// SIMATIC STEP 7 (V5.x) project MK2105
// CPU: CPU 317F-3 PN/DP
// station: 硬件
// station: SINUMERIK
// station: P_ADR_BUS
// program: S7 程序
// program: SINAMICS_In_NCU_710

SYMBOL_TABLE
"ALMSG_DB"	DB 2	UDT 2	// Interface for Alarms & Messages
"gp_par"	DB 7	FB 1	// Parameters for Baseprogram
"NC"	DB 10	UDT 10	// Interface NC
"BAG"	DB 11	UDT 11	// Interface for BAG
"PI"	DB 16	DB 16	// Datainterface PI-Services
"SPL"	DB 18	DB 18	// SPL dataarea
"MMC"	DB 19	UDT 19	// Interface MMC-Signals
"Chan1"	DB 21	UDT 21	// Interface for Channel 1
"X"	DB 31	UDT 31	// Interface Axis 1
"Z"	DB 32	UDT 31	// Interface Axis 2
"C"	DB 33	UDT 31	// Interface Axis 3
"A"	DB 34	UDT 31	// Interface Axis 4
"V"	DB 35	UDT 31	// Interface Axis 5
"W"	DB 36	UDT 31	// Interface Axis 6
"TMLoadIF"	DB 71	UDT 71	// Interface for Loading Station (Toolmanag.)
"TMSpindleIF"	DB 72	UDT 72	// Interface Spindle for Toolmanagment
"TMRevIF"	DB 73	UDT 73	// Interface Revolver (Toolmanagment)
"READ_DB0"	DB 100	DB 100	// Read nc data block0
"READ_DB2"	DB 102	DB 102	// Read nc data R296----R299
"Program_Select"	DB 103	DB 103	// Save PLC Select SUB Programe name
"READ_DB3"	DB 104	DB 104	// Read nc data block3
"X_BACK"	DB 106	DB 106	// X_BACK
"SYSTEM_DB"	DB 110	DB 110	// Read system date and time
"USER_DB0"	DB 120	DB 120	// User define data block0
"USER_DB1"	DB 121	DB 121	// User define data block1
"USER_DB2"	DB 122	DB 122	// User define data block2
"USER_DB3"	DB 123	DB 123	// User define data block3
"USER_DB4"	DB 124	DB 124	// User define data block4
"USER_DB5"	DB 125	DB 125	// User define data block5
"USER_DB6"	DB 126	DB 126	// User define data block6
"USER_DB7"	DB 127	DB 127	// User define data block7
"USER_DB8"	DB 128	DB 128	// User define data block8
"USER_DB9"	DB 129	DB 129	// User define data block9
"CtrlE"	DB 1000	DB 1000	// Interface Ctrl-Energy
"SentronPac"	DB 1001	DB 1001	// Interface SentronPac
"ISM_TS"	DB 1002	DB 1002	// Spindle temperature sensor interface
"TMLoadIF_MT"	DB 1071	UDT 1071	// Interface for Loading Station (Multitool)
"TMSpindleIF_MT"	DB 1072	UDT 1072	// Interface for spindle (Multitool)
"TMRevIF_MT"	DB 1073	UDT 1073	// Interface for Revolver (Multitool)
"RUN_UP"	FB 1	FB 1	// Startup Baseprogram
"GET"	FB 2	FB 2	// read NC Variable
"PUT"	FB 3	FB 3	// write NC Variable
"PI_SERV"	FB 4	FB 4	// PI-Services 1
"GETGUD"	FB 5	FB 5	// read GUD-Variable
"PI_SERV2"	FB 7	FB 7	// PI-Services 2
"M2N"	FB 9	FB 9	// Several OPs/NCUs
"SI_Relais"	FB 10	FB 10	// Safety Integrated: Relais
"SI_BrakeTest"	FB 11	FB 11	// Safety Integrated: Brake Test
"Diagnose"	FB 29	FB 29	// Signal recorder and data trigger diagnostics
"GP_HP"	FC 2	FC 2	// cyclic Baseprogram
"GP_PRAL"	FC 3	FC 3	// alarmtriggered Baseprogram
"GP_DIAG"	FC 5	FC 5	// Diagnosis alarm and Modul failure
"TM_TRANS2"	FC 6	FC 6	// Transfer for Toolmanagment (Multitool)
"TM_REV"	FC 7	FC 7	// Transfer for Revolverchange
"TM_TRANS"	FC 8	FC 8	// Transfer for Toolmanagment
"ASUP"	FC 9	FC 9	// asynchronous Subprograms
"AL_MSG"	FC 10	FC 10	// Alarms & Messages
"BHGDisp"	FC 13	FC 13	// Displaycontrol for Handheld Unit
"YDelta"	FC 17	FC 17	// Y / Delta Control
"SpinCtrl"	FC 18	FC 18	// Spindlecontrol / Part-, Positioning-axis
"MCP_IFM"	FC 19	FC 19	// MCP-Signals to Interface, Variant M
"Transfer"	FC 21	FC 21	// Quick Datachannel
"TM_DIR"	FC 22	FC 22	// Directioncontrol for Toolmanagment Mag.
"MCP_IFM2"	FC 24	FC 24	// MCP-Signals to Interface, Variant small
"MCP_IFT"	FC 25	FC 25	// MCP-Signals to Interface, Variant T
"HPU_MCP"	FC 26	FC 26	// MCP-Signals of PHG to Interface
"Functions block call"	FC 29	FC 29	// Call all functions blocks
"Enable_Control"	FC 30	FC 30
"All motors_ control"	FC 31	FC 31
"NC AND PLC CHANGE DATA"	FC 32	FC 32
"HandWheelUnit_Control"	FC 33	FC 33
"Grinding_Speed_1"	FC 34	FC 34
"Select program"	FC 35	FC 35
"HandWheel_Control"	FC 36	FC 36
"Single Key control"	FC 37	FC 37
"Axis_Control"	FC 38	FC 38
"System_Date"	FC 39	FC 39
"X_BACK_Control"	FC 40	FC 40
"Grinding_Speed_2"	FC 41	FC 41
"Truss manipulator"	FC 42	FC 42
"Auto_Key"	I 0.0	BOOL
"MDA_Key"	I 0.1	BOOL
"TEACH_Key"	I 0.2	BOOL
"JOG_Key"	I 0.3	BOOL
"INC1_Key"	I 1.0	BOOL
"INC10_Key"	I 1.1	BOOL
"INC100_Key"	I 1.2	BOOL
"INC1000_Key"	I 1.3	BOOL
"INC10000_Key"	I 1.4	BOOL
"INC_VAR_Key"	I 1.5	BOOL
"Refpoint_Key"	I 1.6	BOOL
"Repos_Key"	I 1.7	BOOL
"Nc_Stop"	I 2.0	BOOL
"Nc_Start"	I 2.1	BOOL
"Drive_Unable_Key"	I 2.2	BOOL
"Drive_Enable_Key"	I 2.3	BOOL
"Spindle_Unable_Key"	I 2.4	BOOL
"Spindle_Enable_Key"	I 2.5	BOOL
"Key_Pos2"	I 2.6	BOOL
"Key_Pos0"	I 2.7	BOOL
"Feed_A"	I 3.0	BOOL
"Feed_B"	I 3.1	BOOL
"Feed_C"	I 3.2	BOOL
"Feed_D"	I 3.3	BOOL
"Feed_E"	I 3.4	BOOL
"Key_Pos1"	I 3.6	BOOL
"Reset_Key"	I 3.7	BOOL
"R10_手动对刀"	I 4.0	BOOL
"7th_气动门1"	I 4.1	BOOL
"A_axis"	I 4.2	BOOL
"X_axis"	I 4.3	BOOL
"Key_Pos3"	I 4.4	BOOL
"Rapid_Key"	I 4.5	BOOL
"-_Key"	I 4.6	BOOL
"+_Key"	I 4.7	BOOL
"W_axis"	I 5.0	BOOL
"8th_气动门2"	I 5.1	BOOL
"9th_气动门锁强开"	I 5.2	BOOL
"R11_自动对刀"	I 5.3	BOOL
"R12_工件坐标"	I 5.4	BOOL
"V_axis"	I 5.5	BOOL
"C_axis"	I 5.6	BOOL
"Z_axis"	I 5.7	BOOL
"T15_照明"	I 6.1	BOOL
"T14_机械门锁"	I 6.2	BOOL
"T13_X轴快退"	I 6.3	BOOL
"T12_润滑"	I 6.4	BOOL
"T11_吸雾"	I 6.5	BOOL
"T10_Һѹ"	I 6.6	BOOL
"T9_冷却3"	I 6.7	BOOL
"T8_冷却2"	I 7.0	BOOL
"T7_冷却1"	I 7.1	BOOL
"T6_空调"	I 7.2	BOOL
"T5_滚轮"	I 7.3	BOOL
"T4_砂轮"	I 7.4	BOOL
"T3_"	I 7.5	BOOL
"T2_修整"	I 7.6	BOOL
"T1_DRF"	I 7.7	BOOL
"KT1_X51.1_L1"	I 10.0	BOOL	// 轴选输入1
"KT2_X51.2_L2"	I 10.1	BOOL	// 轴选输入2
"KT3_X51.3_L4"	I 10.2	BOOL	// 轴选输入3
"KT4_X52.1_R1"	I 10.3	BOOL	// 倍率输入1
"KT5_X52.2_R2"	I 10.4	BOOL	// 倍率输入2
"KT6_X52.3_R4"	I 10.5	BOOL	// 倍率输入3
"KT7_X55.1"	I 10.6	BOOL
"KT8_X55.2"	I 10.7	BOOL
"KT9_X55.5"	I 11.0	BOOL
"-SB0_急停按钮"	I 32.0	BOOL	// 急停按钮输入(SB0)
"-SQ1_X+"	I 32.1	BOOL	// X轴正限位(SQ1)
"-SQ2_X-"	I 32.2	BOOL	// X轴负限位(SQ2)
"-SQ3_Z+"	I 32.3	BOOL	// Z轴正限位(SQ3)
"-SQ4_Z-"	I 32.4	BOOL	// Z轴负限位(SQ4)
"-ALARM_制动单元报警"	I 32.5	BOOL	// 砂轮主轴变频器制动单元报警
"-QF1_润滑泵"	I 32.6	BOOL	// 润滑泵过载保护(QF1)
"-KP_润滑油液位检测"	I 32.7	BOOL	// 润滑油液位检测(KP1)
"-QF2_液压泵"	I 33.0	BOOL	// 液压泵过载保护(QF2)
"-KP_液压油压力检测"	I 33.1	BOOL	// 液压油压力检测(KP2)
"-QF3_冷却泵1"	I 33.2	BOOL	// 冷却泵1过载保护(QF3)
"-QF4_冷却泵2"	I 33.3	BOOL	// 冷却泵2过载保护(QF4)
"-QF5_冷却泵3"	I 33.4	BOOL	// 冷却泵3过载保护(QF5)
"-QF6_吸雾器"	I 33.5	BOOL	// 吸雾器过载保护(QF6)
"-QF7_水冷机"	I 33.6	BOOL	// 水冷机过载保护(QF7)
"-ALARM_水冷机报警"	I 33.7	BOOL	// 水冷机报警(ALARM1)
"-QF8_电柜空调"	I 34.0	BOOL	// 电箱空调过载保护(QF8)
"-ALARM_空调报警"	I 34.1	BOOL	// 电箱空调报警(ALARM2)
"-QF9_冷却装置"	I 34.2	BOOL	// 冷却装置过载保护(QF9)
"-KP_冷却油液位检测"	I 34.3	BOOL	// 冷却油液位检测(KP3)
"-QF10_直流电源"	I 34.4	BOOL	// 直流电源过载保护(QF10)
"-QF11_控制变压器"	I 34.5	BOOL	// 控制变压器过载保护(QF11)
"-QF14_砂轮电机"	I 34.6	BOOL	// 砂轮电机变频器过载保护(QF14)
"-ALARM_主轴变频器报警"	I 34.7	BOOL	// 砂轮电机变频器报警(ALARM3)
"-QF15_滚轮电机"	I 35.0	BOOL	// 滚轮电机驱动器过载保护(QF15)
"-ALARM_滚轮驱动器报警"	I 35.1	BOOL	// 滚轮电机驱动器报警(ALARM4)
"-QF16_AR润滑泵"	I 35.2	BOOL	// AR润滑泵过载保护(QF16)
"OFF1_Ready"	I 35.3	BOOL	// OFF1_Ready
"EP_Ready"	I 35.4	BOOL	// EP_Ready
"-SQ5_卡盘松开到位"	I 35.5	BOOL	// 液压卡盘松开到位(SQ5)
"-SQ6_卡盘夹紧到位"	I 35.6	BOOL	// 液压卡盘夹紧到位(SQ6)
"-KP_气压检测"	I 35.7	BOOL	// 机床气压检测(KP4)
"-SQ7_左门1打开到位"	I 36.0	BOOL	// 左防护门1打开到位(SQ7)
"-SQ8_左门1关闭到位"	I 36.1	BOOL	// 左防护门1关闭到位(SQ8)
"-SQ9_右门1打开到位"	I 36.2	BOOL	// 右防护门1打开到位(SQ9)
"-SQ10_右门1关闭到位"	I 36.3	BOOL	// 右防护门1关闭到位(SQ10)
"-SQ11_左门2打开到位"	I 36.4	BOOL	// 左防护门2打开到位(SQ11)
"-SQ12_左门2关闭到位"	I 36.5	BOOL	// 左防护门2关闭到位(SQ12)
"-SQ13_右门2打开到位"	I 36.6	BOOL	// 右防护门2打开到位(SQ13)
"-SQ14_右门2关闭到位"	I 36.7	BOOL	// 右防护门2关闭到位(SQ14)
"-ALARM_主轴温度报警"	I 37.0	BOOL	// 砂轮电机温度报警(ALARM5)
"-QF17_驱动电源"	I 37.1	BOOL	// 驱动器电源过载保护(QF17)
"-KP_润滑液位检测"	I 37.2	BOOL	// 润滑油液位检测
"-KP_水冷回路检测1"	I 37.3	BOOL	// 水冷回路检测1
"-KP_水冷回路检测2"	I 37.4	BOOL	// 水冷回路检测2
"-KP_水冷回路检测3"	I 37.5	BOOL	// 水冷回路检测3
"-KP_水冷回路检测4"	I 37.6	BOOL	// 水冷回路检测4
"-KP_润滑气压检测"	I 37.7	BOOL	// 润滑气压检测
"-SF_脚踩开关"	I 38.0	BOOL	// 脚踩开关(SF)
"-LCCK_门锁状态1"	I 38.1	BOOL	// 机械门锁状态1
"-LCCK_门锁状态2"	I 38.2	BOOL	// 机械门锁状态2
"-LCCK_门锁状态3"	I 38.3	BOOL	// 机械门锁状态3
"-UPS_电池供电"	I 38.4	BOOL	// UPS电池供电
"-UPS_电池报警"	I 38.5	BOOL	// UPS电池状态(ready or no)
"-UPS_>80%负荷"	I 38.6	BOOL	// UPS电源>80%负荷
"-KP_漏油检测"	I 38.7	BOOL	// 冷却油箱漏油检测
"-KP_灭火装置"	I 39.0	BOOL	// 灭火装置状态检测
"-KP_光幕1"	I 39.1	BOOL	// 光幕状态1
"-KP_光幕2"	I 39.2	BOOL	// 光幕状态2
"-SB1_辅助急停1"	I 39.3	BOOL	// 辅助急停1(-SB1)
"-SB2_辅助急停2"	I 39.4	BOOL	// 辅助急停2(-SB2)
"-KP_水冷回路检测5"	I 39.5	BOOL	// 水冷回路检测5
"-KP_水冷回路检测6"	I 39.6	BOOL	// 水冷回路检测6
"-KP_电主轴水冷回路检测"	I 39.7	BOOL	// 电主轴水冷回路检测
"Input1_取成品到位"	I 40.0	BOOL	// 机械手取成品到位
"Input2_送毛坯到位"	I 40.1	BOOL	// 机械手送毛坯到位
"Input3_夹爪回到位"	I 40.2	BOOL	// 机械手夹爪回到位
"Input4_备用1"	I 40.3	BOOL
"Input5_备用2"	I 40.4	BOOL
"Input6_备用3"	I 40.5	BOOL
"Input7_备用4"	I 40.6	BOOL
"Input8_备用5"	I 40.7	BOOL
"Spindle_Override"	IB 0	BYTE
"Feed_Ovwerride"	IB 3	BYTE
"ZERO"	M 0.0	BOOL	// Constant "0"
"ONE"	M 0.1	BOOL	// Constant "1"
"Feed_Enable_X"	M 0.2	BOOL
"X_Ref_OK"	M 0.3	BOOL
"X_break_On"	M 0.4	BOOL
"Feed_Enable_Z"	M 0.5	BOOL
"Z_Ref_OK"	M 0.6	BOOL
"Z_break_On"	M 0.7	BOOL
"Feed_Enable_C"	M 1.0	BOOL
"C_Ref_OK"	M 1.1	BOOL
"C_break_On"	M 1.2	BOOL
"Feed_Enable_A"	M 1.3	BOOL
"A_Ref_OK"	M 1.4	BOOL
"A_break_On"	M 1.5	BOOL
"Feed_Enable_V"	M 1.6	BOOL
"V_Ref_OK"	M 1.7	BOOL
"V_break_On"	M 2.0	BOOL
"Feed_Enable_W"	M 2.1	BOOL
"W_Ref_OK"	M 2.2	BOOL
"W_break_On"	M 2.3	BOOL
"Spindle_Enable"	M 2.6	BOOL
"SpindleOverrid_Disable"	M 2.7	BOOL
"*X"	M 3.0	BOOL
"*Z"	M 3.1	BOOL
"*C"	M 3.2	BOOL
"*A"	M 3.3	BOOL
"*V"	M 3.4	BOOL
"*W"	M 3.5	BOOL
"*HHU"	M 3.6	BOOL
"*1"	M 4.0	BOOL
"*10"	M 4.1	BOOL
"*100"	M 4.2	BOOL
"Key_0"	M 10.0	BOOL
"Key_1"	M 10.1	BOOL
"Key_2"	M 10.2	BOOL
"Key_3"	M 10.3	BOOL
"EMG_Active"	M 21.2	BOOL
"Chan1_Stop"	M 21.7	BOOL
"Time_Lock_Active"	M 153.6	BOOL
"EMG_FP"	M 500.3	BOOL	// 松开急停上升沿脉冲
"HHU_FN"	M 500.5	BOOL	// 关断手持下降沿脉冲
"ONE_FP"	M 500.7	BOOL	// 上电上升沿脉冲
"Auto_LED"	Q 0.0	BOOL	// Auto operation mode active indicator light
"MDA_LED"	Q 0.1	BOOL	// MDA operation mode active indicator light
"TEACH_LED"	Q 0.2	BOOL	// TEACH operation mode active indicator light
"JOG_LED"	Q 0.3	BOOL	// JOG operation mode active indicator light
"INC_1_LED"	Q 0.4	BOOL	// INC 1 active indicator light
"INC_10_LED"	Q 0.5	BOOL	// INC 10 active indicator light
"INC_100_LED"	Q 0.6	BOOL	// INC 100 active indicator light
"INC_1000_LED"	Q 0.7	BOOL	// INC 1000 active indicator light
"INC_10000_LED"	Q 1.0	BOOL	// INC 10000 active indicator light
"INC_VAR_LED"	Q 1.1	BOOL	// INC VAR active indicator light
"REF_LED"	Q 1.2	BOOL	// REF operation mode active indicator light
"REPOS_LED"	Q 1.3	BOOL	// Repos operation mode active indicator light
"NCSTART_LED"	Q 1.4	BOOL	// NC start active indicator light
"NCSTOP_LED"	Q 1.5	BOOL	// NC stop active indicator light
"FeedDisable_LED"	Q 1.6	BOOL	// Feed disable indicator light
"FeedEnable_LED"	Q 1.7	BOOL	// Feed enable active indicator light
"SpindleDisable_LED"	Q 2.0	BOOL	// Spindle disable indicator light
"SpindleEnable_LED"	Q 2.1	BOOL	// Spindle enable active indicator light
"SingleBlock_LED"	Q 2.2	BOOL	// Single operation mode active indicator light
"R10_LED_手动对刀"	Q 2.3	BOOL	// 手动对刀有效
"7th_LED_气动门1"	Q 2.4	BOOL	// 气动门1打开
"A_LED"	Q 2.5	BOOL	// The A axis be selected indicator light
"X_LED"	Q 2.6	BOOL	// The X axis be selected indicator light
"-_LED"	Q 2.7	BOOL
"+_LED"	Q 3.0	BOOL
"W_LED"	Q 3.1	BOOL	// The W axis be selected indicator light
"8th_LED_气动门2"	Q 3.2	BOOL	// 气动门2打开
"9th_LED_强制打开"	Q 3.3	BOOL	// 气动门强制打开有效
"R11_LED_自动对刀"	Q 3.4	BOOL	// 自动对刀有效
"R12_LED_工件坐标"	Q 3.5	BOOL	// 工件坐标系有效
"V_LED"	Q 3.6	BOOL	// The V axis be selected indicator light
"C_LED"	Q 3.7	BOOL	// The C axis be selected indicator light
"Z_LED"	Q 4.0	BOOL	// The Z axis be selected indicator light
"T15_LED_照明"	Q 4.1	BOOL	// 机床照明灯燃亮
"T14_LED_机械锁"	Q 4.2	BOOL	// 机械门锁打开
"T13_LED_X轴快退"	Q 4.3	BOOL	// X轴快退
"T12_LED_润滑"	Q 4.4	BOOL	// 机床润滑泵启动
"T11_LED_吸雾"	Q 4.5	BOOL	// 吸雾器启动
"T10_LED_Һѹ"	Q 4.6	BOOL	// 液压泵启动
"T9_LED_冷却3"	Q 4.7	BOOL	// 冷却泵3启动
"T8_LED_冷却2"	Q 5.0	BOOL	// 冷却泵2启动
"T7_LED_冷却1"	Q 5.1	BOOL	// 冷却泵1启动
"T6_LED_空调"	Q 5.2	BOOL	// 电箱空调启动
"T5_LED_滚轮"	Q 5.3	BOOL	// 滚轮电机启动
"T4_LED_砂轮"	Q 5.4	BOOL	// 砂轮电机启动
"T3_LED_"	Q 5.5	BOOL
"T2_LED_修整"	Q 5.6	BOOL	// 砂轮修整有效
"T1_LED_DRF"	Q 5.7	BOOL	// 手轮干涉有效
"KT_OUT1_X53.1"	Q 7.0	BOOL	// 手轮干涉有效
"KT_OUT2_X53.2"	Q 7.1	BOOL
"KT_OUT3_X53.3"	Q 7.2	BOOL
"KT_OUT4_X54.1"	Q 7.3	BOOL
"KT_OUT5_X54.2"	Q 7.4	BOOL
"KT_OUT6_X54.3"	Q 7.5	BOOL
"KA1_9_48"	Q 32.0	BOOL	// 9_48 run/off output control(KA1)
"KA2_9_63"	Q 32.1	BOOL	// 9_63 run/off output control(KA2)
"KA3_9_64"	Q 32.2	BOOL	// 9_64 run/off output control(KA3)
"KA4_导轨润滑"	Q 32.3	BOOL	// 机床润滑泵启动/停止(KA4)
"KA5_液压泵"	Q 32.4	BOOL	// 液压泵启动/停止(KA5)
"KA6_冷却泵1"	Q 32.5	BOOL	// 冷却泵1启动/停止(KA6)
"KA7_冷却泵2"	Q 32.6	BOOL	// 冷却泵2启动/停止(KA7)
"KA8_冷却泵3"	Q 32.7	BOOL	// 冷却泵3启动/停止(KA8)
"KA9_吸雾器"	Q 33.0	BOOL	// 吸雾器启动/停止(KA9)
"KA10_水冷机"	Q 33.1	BOOL	// 水冷机启动/停止(KA10)
"KA11_空调"	Q 33.2	BOOL	// 电箱空调启动/停止(KA11)
"KA12_照明灯"	Q 33.3	BOOL	// 机床照明灯燃亮/熄灭(KA12)
"KA13_卡盘夹紧"	Q 33.4	BOOL	// 液压卡盘夹紧(KA13)
"KA14_卡盘松开"	Q 33.5	BOOL	// 液压卡盘松开(KA14)
"KA15_卸荷阀"	Q 33.6	BOOL	// 卸荷阀打开/关闭(KA15)
"KA16_砂轮启停"	Q 33.7	BOOL	// 砂轮电机启动/停止(KA16)
"KA17_滚轮使能"	Q 34.0	BOOL	// 滚轮驱动使能(KA17)
"KA18_报警复位"	Q 34.1	BOOL	// 滚轮驱动器报警复位(KA18)
"KA19_滚轮启停"	Q 34.2	BOOL	// 滚轮电机启动/停止(KA19)
"KA20_红色"	Q 34.3	BOOL	// 红色警示灯燃亮/熄灭(KA20)
"KA21_黄色"	Q 34.4	BOOL	// 黄色警示灯燃亮/熄灭(KA21)
"KA22_绿色"	Q 34.5	BOOL	// 绿色警示灯燃亮/熄灭(KA22)
"KA23_门1打开"	Q 34.6	BOOL	// 防护门1打开(KA23)
"KA24_门1关闭"	Q 34.7	BOOL	// 防护门1关闭(KA24)
"KA25_门2打开"	Q 35.0	BOOL	// 防护门2打开(KA25)
"KA26_门2关闭"	Q 35.1	BOOL	// 防护门2关闭(KA26)
"KA27_主轴润滑"	Q 35.2	BOOL	// AR润滑泵启动/停止(KA27)
"KA28_机械门锁"	Q 35.3	BOOL	// 机械门锁打开/锁紧(KA28)
"KA29_主轴气路"	Q 35.4	BOOL	// 电主轴气路控制(KA29)
"KA30_"	Q 35.5	BOOL	// 备用(KA30)
"KA31_"	Q 35.6	BOOL	// 备用(KA31)
"KA32_"	Q 35.7	BOOL	// 备用(KA32)
"KA33_"	Q 36.0	BOOL	// 备用(KA33)
"KA34_"	Q 36.1	BOOL	// 备用(KA34)
"KA35_"	Q 36.2	BOOL	// 备用(KA35)
"KA36_"	Q 36.3	BOOL	// 备用(KA36)
"KA37_"	Q 36.4	BOOL	// 备用(KA37)
"KA38_"	Q 36.5	BOOL	// 备用(KA38)
"KA39_"	Q 36.6	BOOL	// 备用(KA39)
"KA40_"	Q 36.7	BOOL	// 备用(KA40)
"KA41_准备就绪"	Q 37.0	BOOL	// 机械手准备就绪
"KA42_预完成"	Q 37.1	BOOL	// 预完成
"KA43_机械手故障"	Q 37.2	BOOL	// 机械手故障
"KA44_卡盘松开完成"	Q 37.3	BOOL	// 卡盘松开完成
"KA45_卡盘夹紧完成"	Q 37.4	BOOL	// 卡盘夹紧完成
"KA46_备用1"	Q 37.5	BOOL	// 机械手备用(KA46)
"KA47_备用2"	Q 37.6	BOOL	// 机械手备用(KA47)
"KA48_备用3"	Q 37.7	BOOL	// 机械手备用(KA48)
"READ_CLK"	SFC 1	SFC 1	// Read System Clock
"ALARM_SQ"	SFC 17	SFC 17	// Generate Block-Related Messages with Acknowledgment
"TIME_TCK"	SFC 64	SFC 64	// Read the System Time
"KT0"	T 10	TIMER	// 急停报警延时
"KT1"	T 11	TIMER	// System power_on delay(T9_63)
"KT2"	T 12	TIMER	// System power_on delay(T9_64)
"KT3"	T 13	TIMER	// System power_off delay(T9_63)
"KT4"	T 14	TIMER	// System power_off delay(T9_48)
"KT5"	T 15	TIMER	// 报警延时
"KT6"	T 16	TIMER	// 手动对刀状态显示延时1
"KT7"	T 17	TIMER	// 手动对刀状态显示延时2
"KT8"	T 18	TIMER	// 自动对刀状态显示延时1
"KT9"	T 19	TIMER	// 自动对刀状态显示延时2
"KT10"	T 20	TIMER	// 主轴启动主轴润滑及供气初次运行时间
"KT11"	T 21	TIMER	// 主轴润滑状态显示延时1
"KT12"	T 22	TIMER	// 主轴润滑状态显示延时2
"KT13"	T 23	TIMER	// 滚轮使能断延时
"KT14"	T 24	TIMER	// 手动导轨润滑润滑时间
"KT15"	T 25	TIMER	// 自动导轨润滑间歇时间
"KT16"	T 26	TIMER	// 自动导轨润滑润滑时间
"KT17"	T 27	TIMER	// 装载异步子程序脉冲延时
"KT18"	T 28	TIMER	// 手持单元关断延时
"T_ASUP_DELAY1"	T 29	TIMER	// X轴快退沿脉冲延时1
"T_ASUP_DELAY2"	T 30	TIMER	// X轴快退沿脉冲延时2
"T_ASUP_DELAY3"	T 31	TIMER	// X轴快退沿脉冲延时3
"KT22"	T 32	TIMER	// 松开急停后主轴润滑及供气初次运行时间
END_SYMBOL_TABLE

TYPE UDT 2
VERSION : 0.0
  STRUCT
   C1 : STRUCT 	//From Channel 1
    FDD_5100xx : ARRAY  [0 .. 15 ] OF //Feed disable A.no.51000-510015
    BOOL ;
    FDD_RID_5101xx : ARRAY  [0 .. 31 ] OF //Feed and read-in disable A.no.510100-510131
    BOOL ;
    RID_5102xx : ARRAY  [0 .. 31 ] OF //Read-in disable A.no.510200-510231
    BOOL ;
    NCSD_5103xx : ARRAY  [0 .. 15 ] OF //NC start disable A.no.510300-510315
    BOOL ;
    FdStop_1_5111xx : ARRAY  [0 .. 15 ] OF //Feed stop GEOaxis 1 A.no.511100-511115
    BOOL ;
    FdStop_2_5112xx : ARRAY  [0 .. 15 ] OF //Feed stop GEOaxis 2 A.no.511200-511215
    BOOL ;
    FdStop_3_5113xx : ARRAY  [0 .. 15 ] OF //Feed stop GEOaxis 3 A.no.511300-511315
    BOOL ;
   END_STRUCT ;
   C2 : STRUCT 	//From Channel 2
    FDD_5200xx : ARRAY  [0 .. 15 ] OF //Feed disable A.no.520000-520015
    BOOL ;
    FDD_RID_5201xx : ARRAY  [0 .. 31 ] OF //Feed and read-in disable A.no.520100-520131
    BOOL ;
    RID_5202xx : ARRAY  [0 .. 31 ] OF //Read-in disable A.no.520200-520231
    BOOL ;
    NCSD_5203xx : ARRAY  [0 .. 15 ] OF //NC start disable A.no.520300-520315
    BOOL ;
    FdStop_1_5211xx : ARRAY  [0 .. 15 ] OF //Feed stop GEOaxis 1 A.no.521100-521115
    BOOL ;
    FdStop_2_5212xx : ARRAY  [0 .. 15 ] OF //Feed stop GEOaxis 2 A.no.521200-521215
    BOOL ;
    FdStop_3_5213xx : ARRAY  [0 .. 15 ] OF //Feed stop GEOaxis 3 A.no.521300-521315
    BOOL ;
   END_STRUCT ;
   C3 : STRUCT 	//From Channel 3
    FDD_5300xx : ARRAY  [0 .. 15 ] OF //Feed disable A.no.530000-530015
    BOOL ;
    FDD_RID_5301xx : ARRAY  [0 .. 31 ] OF //Feed and read-in disable A.no.530100-530131
    BOOL ;
    RID_5302xx : ARRAY  [0 .. 31 ] OF //Read-in disable A.no.530200-530231
    BOOL ;
    NCSD_5303xx : ARRAY  [0 .. 15 ] OF //NC start disable A.no.530300-530315
    BOOL ;
    FdStop_1_5311xx : ARRAY  [0 .. 15 ] OF //Feed stop GEOaxis 1 A.no.531100-531115
    BOOL ;
    FdStop_2_5312xx : ARRAY  [0 .. 15 ] OF //Feed stop GEOaxis 2 A.no.531200-531215
    BOOL ;
    FdStop_3_5313xx : ARRAY  [0 .. 15 ] OF //Feed stop GEOaxis 3 A.no.531300-531315
    BOOL ;
   END_STRUCT ;
   C4 : STRUCT 	//From Channel 4
    FDD_5400xx : ARRAY  [0 .. 15 ] OF //Feed disable A.no.540000-540015
    BOOL ;
    FDD_RID_5401xx : ARRAY  [0 .. 31 ] OF //Feed and read-in disable A.no.540100-540131
    BOOL ;
    RID_5402xx : ARRAY  [0 .. 31 ] OF //Read-in disable A.no.540200-540231
    BOOL ;
    NCSD_5403xx : ARRAY  [0 .. 15 ] OF //NC start disable A.no.540300-540315
    BOOL ;
    FdStop_1_5411xx : ARRAY  [0 .. 15 ] OF //Feed stop GEOaxis 1 A.no.541100-541115
    BOOL ;
    FdStop_2_5412xx : ARRAY  [0 .. 15 ] OF //Feed stop GEOaxis 2 A.no.541200-541215
    BOOL ;
    FdStop_3_5413xx : ARRAY  [0 .. 15 ] OF //Feed stop GEOaxis 3 A.no.541300-541315
    BOOL ;
   END_STRUCT ;
   C5 : STRUCT 	//From Channel 5
    FDD_5500xx : ARRAY  [0 .. 15 ] OF //Feed disable A.no.550000-550015
    BOOL ;
    FDD_RID_5501xx : ARRAY  [0 .. 31 ] OF //Feed and read-in disable A.no.550100-550131
    BOOL ;
    RID_5502xx : ARRAY  [0 .. 31 ] OF //Read-in disable A.no.550200-550231
    BOOL ;
    NCSD_5503xx : ARRAY  [0 .. 15 ] OF //NC start disable A.no.550300-550315
    BOOL ;
    FdStop_1_5511xx : ARRAY  [0 .. 15 ] OF //Feed stop GEOaxis 1 A.no.551100-551115
    BOOL ;
    FdStop_2_5512xx : ARRAY  [0 .. 15 ] OF //Feed stop GEOaxis 2 A.no.551200-551215
    BOOL ;
    FdStop_3_5513xx : ARRAY  [0 .. 15 ] OF //Feed stop GEOaxis 3 A.no.551300-551315
    BOOL ;
   END_STRUCT ;
   C6 : STRUCT 	//From Channel 6
    FDD_5600xx : ARRAY  [0 .. 15 ] OF //Feed disable A.no.560000-560015
    BOOL ;
    FDD_RID_5601xx : ARRAY  [0 .. 31 ] OF //Feed and read-in disable A.no.560100-560131
    BOOL ;
    RID_5602xx : ARRAY  [0 .. 31 ] OF //Read-in disable A.no.560200-560231
    BOOL ;
    NCSD_5603xx : ARRAY  [0 .. 15 ] OF //NC start disable A.no.560300-560315
    BOOL ;
    FdStop_1_5611xx : ARRAY  [0 .. 15 ] OF //Feed stop GEOaxis 1 A.no.561100-561115
    BOOL ;
    FdStop_2_5612xx : ARRAY  [0 .. 15 ] OF //Feed stop GEOaxis 2 A.no.561200-561215
    BOOL ;
    FdStop_3_5613xx : ARRAY  [0 .. 15 ] OF //Feed stop GEOaxis 3 A.no.561300-561315
    BOOL ;
   END_STRUCT ;
   C7 : STRUCT 	//From Channel 7
    FDD_5700xx : ARRAY  [0 .. 15 ] OF //Feed disable A.no.570000-570015
    BOOL ;
    FDD_RID_5701xx : ARRAY  [0 .. 31 ] OF //Feed and read-in disable A.no.570100-570131
    BOOL ;
    RID_5702xx : ARRAY  [0 .. 31 ] OF //Read-in disable A.no.570200-570231
    BOOL ;
    NCSD_5703xx : ARRAY  [0 .. 15 ] OF //NC start disable A.no.570300-570315
    BOOL ;
    FdStop_1_5711xx : ARRAY  [0 .. 15 ] OF //Feed stop GEOaxis 1 A.no.571100-511115
    BOOL ;
    FdStop_2_5712xx : ARRAY  [0 .. 15 ] OF //Feed stop GEOaxis 2 A.no.571200-511215
    BOOL ;
    FdStop_3_5713xx : ARRAY  [0 .. 15 ] OF //Feed stop GEOaxis 3 A.no.571300-511315
    BOOL ;
   END_STRUCT ;
   C8 : STRUCT 	//From Channel 8
    FDD_5800xx : ARRAY  [0 .. 15 ] OF //Feed disable A.no.580000-580015
    BOOL ;
    FDD_RID_5801xx : ARRAY  [0 .. 31 ] OF //Feed and read-in disable A.no.580100-510131
    BOOL ;
    RID_5802xx : ARRAY  [0 .. 31 ] OF //Read-in disable A.no.580200-580231
    BOOL ;
    NCSD_5803xx : ARRAY  [0 .. 15 ] OF //NC start disable A.no.580300-580315
    BOOL ;
    FdStop_1_5811xx : ARRAY  [0 .. 15 ] OF //Feed stop GEOaxis 1 A.no.581100-511115
    BOOL ;
    FdStop_2_5812xx : ARRAY  [0 .. 15 ] OF //Feed stop GEOaxis 2 A.no.581200-511215
    BOOL ;
    FdStop_3_5813xx : ARRAY  [0 .. 15 ] OF //Feed stop GEOaxis 3 A.no.581300-511315
    BOOL ;
   END_STRUCT ;
   _1FdStop6001xx : ARRAY  [0 .. 15 ] OF //Feed stop axis/spindle 1
   BOOL ;
   _2FdStop6002xx : ARRAY  [0 .. 15 ] OF //Feed stop axis/spindle 2
   BOOL ;
   _3FdStop6003xx : ARRAY  [0 .. 15 ] OF //Feed stop axis/spindle 3
   BOOL ;
   _4FdStop6004xx : ARRAY  [0 .. 15 ] OF //Feed stop axis/spindle 4
   BOOL ;
   _5FdStop6005xx : ARRAY  [0 .. 15 ] OF //Feed stop axis/spindle 5
   BOOL ;
   _6FdStop6006xx : ARRAY  [0 .. 15 ] OF //Feed stop axis/spindle 6
   BOOL ;
   _7FdStop6007xx : ARRAY  [0 .. 15 ] OF //Feed stop axis/spindle 7
   BOOL ;
   _8FdStop6008xx : ARRAY  [0 .. 15 ] OF //Feed stop axis/spindle 8
   BOOL ;
   _9FdStop6009xx : ARRAY  [0 .. 15 ] OF //Feed stop axis/spindle 9
   BOOL ;
   _10FdStop6010xx : ARRAY  [0 .. 15 ] OF //Feed stop axis/spindle 10
   BOOL ;
   _11FdStop6011xx : ARRAY  [0 .. 15 ] OF //Feed stop axis/spindle 11
   BOOL ;
   _12FdStop6012xx : ARRAY  [0 .. 15 ] OF //Feed stop axis/spindle 12
   BOOL ;
   _13FdStop6013xx : ARRAY  [0 .. 15 ] OF //Feed stop axis/spindle 13
   BOOL ;
   _14FdStop6014xx : ARRAY  [0 .. 15 ] OF //Feed stop axis/spindle 14
   BOOL ;
   _15FdStop6015xx : ARRAY  [0 .. 15 ] OF //Feed stop axis/spindle 15
   BOOL ;
   _16FdStop6016xx : ARRAY  [0 .. 15 ] OF //Feed stop axis/spindle 16
   BOOL ;
   _17FdStop6017xx : ARRAY  [0 .. 15 ] OF //Feed stop axis/spindle 17
   BOOL ;
   _18FdStop6018xx : ARRAY  [0 .. 15 ] OF //Feed stop axis/spindle 18
   BOOL ;
   A7000xx : ARRAY  [0 .. 63 ] OF //Alarm 700000-700063 (user area 0)
   BOOL ;
   A7001xx : ARRAY  [0 .. 63 ] OF //Alarm 700100-700163 (user area 1)
   BOOL ;
   A7002xx : ARRAY  [0 .. 63 ] OF //Alarm 700200-700263 (user area 2)
   BOOL ;
   A7003xx : ARRAY  [0 .. 63 ] OF //Alarm 700300-700363 (user area 3)
   BOOL ;
   A7004xx : ARRAY  [0 .. 63 ] OF //Alarm 700400-700463 (user area 4)
   BOOL ;
   A7005xx : ARRAY  [0 .. 63 ] OF //Alarm 700500-700563 (user area 5
   BOOL ;
   A7006xx : ARRAY  [0 .. 63 ] OF //Alarm 700600-700663 (user area 6)
   BOOL ;
   A7007xx : ARRAY  [0 .. 63 ] OF //Alarm 700700-700763 (user area 7)
   BOOL ;
   A7008xx : ARRAY  [0 .. 63 ] OF //Alarm 700800-700863 (user area 8)
   BOOL ;
   A7009xx : ARRAY  [0 .. 63 ] OF //Alarm 700900-700963 (user area 9)
   BOOL ;
  END_STRUCT ;	
END_TYPE

TYPE UDT 10
VERSION : 0.0
  STRUCT
   A_Disabl_Inp1 : BOOL ;	//Disable digi. NCK input 1
   A_Disabl_Inp2 : BOOL ;	//Disable digi. NCK input 2
   A_Disabl_Inp3 : BOOL ;	//Disable digi. NCK input 3
   A_Disabl_Inp4 : BOOL ;	//Disable digi. NCK input 4
   A_Disabl_Inp5 : BOOL ;	//Disable digi. NCK input 5
   A_Disabl_Inp6 : BOOL ;	//Disable digi. NCK input 6
   A_Disabl_Inp7 : BOOL ;	//Disable digi. NCK input 7
   A_Disabl_Inp8 : BOOL ;	//Disable digi. NCK input 8
   A_Set_Inp1 : BOOL ;	//Set digi. NCK input 1
   A_Set_Inp2 : BOOL ;	//Set digi. NCK input 2
   A_Set_Inp3 : BOOL ;	//Set digi. NCK input 3
   A_Set_Inp4 : BOOL ;	//Set digi. NCK input 4
   A_Set_Inp5 : BOOL ;	//Set digi. NCK input 5
   A_Set_Inp6 : BOOL ;	//Set digi. NCK input 6
   A_Set_Inp7 : BOOL ;	//Set digi. NCK input 7
   A_Set_Inp8 : BOOL ;	//Set digi. NCK input 8
   f0_f15 : ARRAY  [0 .. 15 ] OF BOOL ;	//Reserved
   A_Disabl_Out1 : BOOL ;	//Disable digi. NCK output 1
   A_Disabl_Out2 : BOOL ;	//Disable digi. NCK output 2
   A_Disabl_Out3 : BOOL ;	//Disable digi. NCK output 3
   A_Disabl_Out4 : BOOL ;	//Disable digi. NCK output 4
   A_Disabl_Out5 : BOOL ;	//Disable digi. NCK output 5
   A_Disabl_Out6 : BOOL ;	//Disable digi. NCK output 6
   A_Disabl_Out7 : BOOL ;	//Disable digi. NCK output 7
   A_Disabl_Out8 : BOOL ;	//Disable digi. NCK output 8
   A_OvMask_Out1 : BOOL ;	//Overwrite mask of digi. output 1
   A_OvMask_Out2 : BOOL ;	//Overwrite mask of digi. output 2
   A_OvMask_Out3 : BOOL ;	//Overwrite mask of digi. output 3
   A_OvMask_Out4 : BOOL ;	//Overwrite mask of digi. output 4
   A_OvMask_Out5 : BOOL ;	//Overwrite mask of digi. output 5
   A_OvMask_Out6 : BOOL ;	//Overwrite mask of digi. output 6
   A_OvMask_Out7 : BOOL ;	//Overwrite mask of digi. output 7
   A_OvMask_Out8 : BOOL ;	//Overwrite mask of digi. output 8
   A_Set_Out1 : BOOL ;	//Set digi. NCK output 1
   A_Set_Out2 : BOOL ;	//Set digi. NCK output 2
   A_Set_Out3 : BOOL ;	//Set digi. NCK output 3
   A_Set_Out4 : BOOL ;	//Set digi. NCK output 4
   A_Set_Out5 : BOOL ;	//Set digi. NCK output 5
   A_Set_Out6 : BOOL ;	//Set digi. NCK output 6
   A_Set_Out7 : BOOL ;	//Set digi. NCK output 7
   A_Set_Out8 : BOOL ;	//Set digi. NCK output 8
   A_InMask_Out1 : BOOL ;	//Input mask of digi. output 1
   A_InMask_Out2 : BOOL ;	//Input mask of digi. output 2
   A_InMask_Out3 : BOOL ;	//Input mask of digi. output 3
   A_InMask_Out4 : BOOL ;	//Input mask of digi. output 4
   A_InMask_Out5 : BOOL ;	//Input mask of digi. output 5
   A_InMask_Out6 : BOOL ;	//Input mask of digi. output 6
   A_InMask_Out7 : BOOL ;	//Input mask of digi. output 7
   A_InMask_Out8 : BOOL ;	//Input mask of digi. output 8
   MCP1AxisTbl : ARRAY  [1 .. 22 ] OF BYTE  := B#16#1, B#16#2, B#16#3, B#16#4, B#16#5, B#16#6, B#16#7, B#16#8, B#16#9, B#16#A, B#16#B, B#16#C;	//Axis No. Table MCP1
   MCP1MaxAxis : WORD ;	//max. of Axisno, must be smaller or equal gp_par.MaxAxis
   MCP2AxisTbl : ARRAY  [1 .. 22 ] OF BYTE  := B#16#1, B#16#2, B#16#3, B#16#4, B#16#5, B#16#6, B#16#7, B#16#8, B#16#9, B#16#A, B#16#B, B#16#C;	//Axis No. Table MCP2
   MCP2MaxAxis : WORD ;	//max. of Axisno, must be smaller or equal gp_par.MaxAxis
   f56_0 : BOOL ;
   A_EMERGENCY : BOOL ;	//Emergency stop
   A_EMERGENCY_Ackn : BOOL ;	//Acknowledge emergency stop
   f56_3 : BOOL ;
   A_Keyswitch0 : BOOL ;	//Keyswitch position 0
   A_Keyswitch1 : BOOL ;	//Keyswitch position 1
   A_Keyswitch2 : BOOL ;	//Keyswitch position 2
   A_Keyswitch3 : BOOL ;	//Keyswitch position 3
   A_IncInModeGroup : BOOL ;	//INC inputs in mode group area active
   f57_1 : BOOL ;
   f57_2 : BOOL ;
   A_PCshutdown : BOOL ;	//PC shutdown 840Di
   f57_4 : BOOL ;
   f57_5 : BOOL ;
   f57_6 : BOOL ;
   f57_7 : BOOL ;
   A_CollCheckOff : BOOL ;	//Collisions Check Off
   f58_1 : BOOL ;
   f58_2 : BOOL ;
   f58_3 : BOOL ;
   f58_4 : BOOL ;
   f58_5 : BOOL ;
   f58_6 : BOOL ;
   f58_7 : BOOL ;
   f59 : BYTE ;
   E_ActVal_In1 : BOOL ;	//Actual value of digi. NCK input 1
   E_ActVal_In2 : BOOL ;	//Actual value of digi. NCK input 2
   E_ActVal_In3 : BOOL ;	//Actual value of digi. NCK input 3
   E_ActVal_In4 : BOOL ;	//Actual value of digi. NCK input 4
   f60_4 : BOOL ;
   f60_5 : BOOL ;
   f60_6 : BOOL ;
   f60_7 : BOOL ;
   f61_f62 : ARRAY  [61 .. 61 ] OF BYTE ;
   E_Setpoint_Out1 : BOOL ;	//Setpoint of digi. NCK output 1
   E_Setpoint_Out2 : BOOL ;	//Setpoint of digi. NCK output 2
   E_Setpoint_Out3 : BOOL ;	//Setpoint of digi. NCK output 3
   E_Setpoint_Out4 : BOOL ;	//Setpoint of digi. NCK output 4
   E_Setpoint_Out5 : BOOL ;	//Setpoint of digi. NCK output 5
   E_Setpoint_Out6 : BOOL ;	//Setpoint of digi. NCK output 6
   E_Setpoint_Out7 : BOOL ;	//Setpoint of digi. NCK output 7
   E_Setpoint_Out8 : BOOL ;	//Setpoint of digi. NCK output 8
   f65_f67 : ARRAY  [65 .. 66 ] OF BYTE ;
   E_HW1_moved : BYTE ;	//Handwheel 1 moved
   E_HW2_moved : BYTE ;	//Handwheel 2 moved
   E_HW3_moved : BYTE ;	//Handwheel 3 moved
   E_CounterInchMetr : BYTE ;	//Modification counter inch/metric system of units
   E_MCP1AxisValid : BOOL ;	//from HT6
   E_MCP1WCS : BOOL ;	//from HT6
   f72_2 : BOOL ;
   f72_3 : BOOL ;
   f72_4 : BOOL ;
   f72_5 : BOOL ;
   f72_6 : BOOL ;
   E_MCP1AxKeyDisp : BOOL ;	//Mcp1 Axis Key Displayed
   E_MCP2AxisValid : BOOL ;	//from HT6
   E_MCP2WCS : BOOL ;	//from HT6
   f73_2 : BOOL ;
   f73_3 : BOOL ;
   f73_4 : BOOL ;
   f73_5 : BOOL ;
   f73_6 : BOOL ;
   E_MCP2AxKeyDisp : BOOL ;	//Mcp2 Axis Key Displayed
   MCP1AxisFromHMI : ARRAY  [1 .. 6 ] OF BYTE ;	//Axistable from HT6
   MCP2AxisFromHMI : ARRAY  [1 .. 6 ] OF BYTE ;	//Axistable from HT6
   res86 : WORD ;
   res88 : BYTE ;
   res89 : BYTE ;
   epsToPlc : BYTE ;
   epsFromPlc : BYTE ;
   MpiDpOk : BOOL ;	//Slaves on MPI/DP Ok
   DpOk : BOOL ;	//Slaves on DP Ok
   f92_2 : BOOL ;
   f92_3 : BOOL ;
   f92_4 : BOOL ;
   f92_5 : BOOL ;
   f92_6 : BOOL ;
   f92_7 : BOOL ;
   E_CA_AutoMach : BOOL ;	// Disable collision avoidance : AUTO Machine
   E_CA_AutoTools : BOOL ;	// Disable collision avoidance : AUTO Tools
   E_CA_AutoWorkh : BOOL ;	// Disable collision avoidance : AUTO Workholder
   E_CA_AutoWorkp : BOOL ;	// Disable collision avoidance : AUTO Workpieces
   E_CA_JogMach : BOOL ;	// Disable collision avoidance : JOG Machine
   E_CA_JogTools : BOOL ;	// Disable collision avoidance : JOG Tools
   E_CA_JogWorkh : BOOL ;	// Disable collision avoidance : JOG Workholder
   E_CA_JogWorkp : BOOL ;	// Disable collision avoidance : JOG Workpieces
   f94 : BYTE ;
   f95 : BYTE ;
   E_LanguageID : BYTE ;	// LanguageID on HMI
   E_Chan_HW1_A : BOOL ;	//Channel number for handwheel1 A
   E_Chan_HW1_B : BOOL ;	//Channel number for handwheel1 B
   E_Chan_HW1_C : BOOL ;	//Channel number for handwheel1 C
   E_Chan_HW1_D : BOOL ;	//Channel number for handwheel1 D
   f97_4 : BOOL ;
   f97_5 : BOOL ;
   f97_6 : BOOL ;
   f97_7 : BOOL ;
   E_Chan_HW2_A : BOOL ;	//Channel number for handwheel2 A
   E_Chan_HW2_B : BOOL ;	//Channel number for handwheel2 B
   E_Chan_HW2_C : BOOL ;	//Channel number for handwheel2 C
   E_Chan_HW2_D : BOOL ;	//Channel number for handwheel2 D
   f98_4 : BOOL ;
   f98_5 : BOOL ;
   f98_6 : BOOL ;
   f98_7 : BOOL ;
   E_Chan_HW3_A : BOOL ;	//Channel number for handwheel3 A
   E_Chan_HW3_B : BOOL ;	//Channel number for handwheel3 B
   E_Chan_HW3_C : BOOL ;	//Channel number for handwheel3 C
   E_Chan_HW3_D : BOOL ;	//Channel number for handwheel3 D
   f99_4 : BOOL ;
   f99_5 : BOOL ;
   f99_6 : BOOL ;
   f99_7 : BOOL ;
   E_Ax_A_HW1 : BOOL ;	//Axis number for handwheel1 A
   E_Ax_B_HW1 : BOOL ;	//Axis number for handwheel1 B
   E_Ax_C_HW1 : BOOL ;	//Axis number for handwheel1 C
   E_Ax_D_HW1 : BOOL ;	//Axis number for handwheel1 D
   E_Ax_E_HW1 : BOOL ;	//Axis number for handwheel1 E
   E_CHW_sel1 : BOOL ;	//Contour handwheel selected
   E_HW_sel1 : BOOL ;	//Handwheel selected
   E_Mach_Ax1 : BOOL ;	//Machine axis
   E_Ax_A_HW2 : BOOL ;	//Axis number for handwheel2 A
   E_Ax_B_HW2 : BOOL ;	//Axis number for handwheel2 B
   E_Ax_C_HW2 : BOOL ;	//Axis number for handwheel2 C
   E_Ax_D_HW2 : BOOL ;	//Axis number for handwheel2 D
   E_Ax_E_HW2 : BOOL ;	//Axis number for handwheel2 E
   E_CHW_sel2 : BOOL ;	//Contour handwheel selected
   E_HW_sel2 : BOOL ;	//Handwheel selected
   E_Mach_Ax2 : BOOL ;	//Machine axis
   E_Ax_A_HW3 : BOOL ;	//Axis number for handwheel3 A
   E_Ax_B_HW3 : BOOL ;	//Axis number for handwheel3 B
   E_Ax_C_HW3 : BOOL ;	//Axis number for handwheel3 C
   E_Ax_D_HW3 : BOOL ;	//Axis number for handwheel3 D
   E_Ax_E_HW3 : BOOL ;	//Axis number for handwheel3 E
   E_CHW_sel3 : BOOL ;	//Contour handwheel selected
   E_HW_sel3 : BOOL ;	//Handwheel selected
   E_Mach_Ax3 : BOOL ;	//Machine axis
   E_RemDiag : BOOL ;	//Remote Diagnostic
   f103_1 : BOOL ;
   f103_2 : BOOL ;
   f103_3 : BOOL ;
   f103_4 : BOOL ;
   E_ATready : BOOL ;	//AT-box ready
   E_MMCTemp : BOOL ;	//MMC temperature limit
   E_MMCBatt : BOOL ;	//MMC 101/102 battery alarm
   E_MCP1ready : BOOL ;	//MCP1 ready;
   E_MCP2ready : BOOL ;	//MCP2 ready;
   E_BHGready : BOOL ;	//BHG ready;
   f104_3 : BOOL ;
   f104_4 : BOOL ;
   f104_5 : BOOL ;
   E_FirstOB1 : BOOL ;	//This bit is on for the first OB1 cycle
   E_NCKready : BOOL ;	//NCK CPU ready
   E_CancelToolCmd : BOOL ;	//Terminate canceled tool command
   f105_1 : BOOL ;
   f105_2 : BOOL ;
   f105_3 : BOOL ;
   f105_4 : BOOL ;
   f105_5 : BOOL ;
   f105_6 : BOOL ;
   f105_7 : BOOL ;
   E_CollCheckOff : BOOL ;	//CollisionsCheck Off
   E_EMSTOP : BOOL ;	//EMERGENCY STOP active
   f106_2 : BOOL ;
   f106_3 : BOOL ;
   f106_4 : BOOL ;
   f106_5 : BOOL ;
   f106_6 : BOOL ;
   f106_7 : BOOL ;
   E_InspProbe1 : BOOL ;	//Inspection probe 1 actuated
   E_InspProbe2 : BOOL ;	//Inspection probe 2 actuated
   f107_2 : BOOL ;
   f107_3 : BOOL ;
   f107_4 : BOOL ;
   f107_5 : BOOL ;
   E_NCU_LinkActive : BOOL ;	//NCU link active
   E_SystemInchDim : BOOL ;	//System inch dimension
   f108_0 : BOOL ;
   E_MMC2Ready : BOOL ;	//MMC2-CPU ready
   E_MMCMPIready : BOOL ;	//MMC1-CPU on MPI ready
   E_MMCBTSSready : BOOL ;	//MMC1-CPU on BTSS ready
   f108_4 : BOOL ;
   E_DrivesInCylOp : BOOL ;	//Drives in cylindric operation
   E_611Dready : BOOL ;	//611D ready
   E_NCready : BOOL ;
   E_NCKalarm : BOOL ;	//NCK alarm present
   f109_1 : BOOL ;
   f109_2 : BOOL ;
   f109_3 : BOOL ;
   A_PC_OSfault : BOOL ;	//PC operating system fault, 840Di
   E_HTempAlarm : BOOL ;	//Heat sink temperature alarm NCU 573
   E_ATempAlarm : BOOL ;	//Air temperature alarm
   E_BattAlarm : BOOL ;	//NCK battery alarm
   E_SWCamMinus : ARRAY  [0 .. 31 ] OF BOOL ;	//Software cams minus [0..31]
   E_SWCamPlus : ARRAY  [0 .. 31 ] OF BOOL ;	//Software cams plus [0..31]
   f118_f121 : ARRAY  [0 .. 3 ] OF BYTE ;
   A_Disabl_Inp9 : BOOL ;	//Disable digi. NCK input 9
   A_Disabl_Inp10 : BOOL ;	//Disable digi. NCK input 10
   A_Disabl_Inp11 : BOOL ;	//Disable digi. NCK input 11
   A_Disabl_Inp12 : BOOL ;	//Disable digi. NCK input 12
   A_Disabl_Inp13 : BOOL ;	//Disable digi. NCK input 13
   A_Disabl_Inp14 : BOOL ;	//Disable digi. NCK input 14
   A_Disabl_Inp15 : BOOL ;	//Disable digi. NCK input 15
   A_Disabl_Inp16 : BOOL ;	//Disable digi. NCK input 16
   A_Set_Inp9 : BOOL ;	//Set digi. NCK input 9
   A_Set_Inp10 : BOOL ;	//Set digi. NCK input 10
   A_Set_Inp11 : BOOL ;	//Set digi. NCK input 11
   A_Set_Inp12 : BOOL ;	//Set digi. NCK input 12
   A_Set_Inp13 : BOOL ;	//Set digi. NCK input 13
   A_Set_Inp14 : BOOL ;	//Set digi. NCK input 14
   A_Set_Inp15 : BOOL ;	//Set digi. NCK input 15
   A_Set_Inp16 : BOOL ;	//Set digi. NCK input 16
   A_Disabl_Inp17 : BOOL ;	//Disable digi. NCK input 17
   A_Disabl_Inp18 : BOOL ;	//Disable digi. NCK input 18
   A_Disabl_Inp19 : BOOL ;	//Disable digi. NCK input 19
   A_Disabl_Inp20 : BOOL ;	//Disable digi. NCK input 20
   A_Disabl_Inp21 : BOOL ;	//Disable digi. NCK input 21
   A_Disabl_Inp22 : BOOL ;	//Disable digi. NCK input 22
   A_Disabl_Inp23 : BOOL ;	//Disable digi. NCK input 23
   A_Disabl_Inp24 : BOOL ;	//Disable digi. NCK input 24
   A_Set_Inp17 : BOOL ;	//Set digi. NCK input 17
   A_Set_Inp18 : BOOL ;	//Set digi. NCK input 18
   A_Set_Inp19 : BOOL ;	//Set digi. NCK input 19
   A_Set_Inp20 : BOOL ;	//Set digi. NCK input 20
   A_Set_Inp21 : BOOL ;	//Set digi. NCK input 21
   A_Set_Inp22 : BOOL ;	//Set digi. NCK input 22
   A_Set_Inp23 : BOOL ;	//Set digi. NCK input 23
   A_Set_Inp24 : BOOL ;	//Set digi. NCK input 24
   A_Disabl_Inp25 : BOOL ;	//Disable digi. NCK input 25
   A_Disabl_Inp26 : BOOL ;	//Disable digi. NCK input 26
   A_Disabl_Inp27 : BOOL ;	//Disable digi. NCK input 27
   A_Disabl_Inp28 : BOOL ;	//Disable digi. NCK input 28
   A_Disabl_Inp29 : BOOL ;	//Disable digi. NCK input 29
   A_Disabl_Inp30 : BOOL ;	//Disable digi. NCK input 30
   A_Disabl_Inp31 : BOOL ;	//Disable digi. NCK input 31
   A_Disabl_Inp32 : BOOL ;	//Disable digi. NCK input 32
   A_Set_Inp25 : BOOL ;	//Set digi. NCK input 25
   A_Set_Inp26 : BOOL ;	//Set digi. NCK input 26
   A_Set_Inp27 : BOOL ;	//Set digi. NCK input 27
   A_Set_Inp28 : BOOL ;	//Set digi. NCK input 28
   A_Set_Inp29 : BOOL ;	//Set digi. NCK input 29
   A_Set_Inp30 : BOOL ;	//Set digi. NCK input 30
   A_Set_Inp31 : BOOL ;	//Set digi. NCK input 31
   A_Set_Inp32 : BOOL ;	//Set digi. NCK input 32
   A_Disabl_Inp33 : BOOL ;	//Disable digi. NCK input 33
   A_Disabl_Inp34 : BOOL ;	//Disable digi. NCK input 34
   A_Disabl_Inp35 : BOOL ;	//Disable digi. NCK input 35
   A_Disabl_Inp36 : BOOL ;	//Disable digi. NCK input 36
   A_Disabl_Inp37 : BOOL ;	//Disable digi. NCK input 37
   A_Disabl_Inp38 : BOOL ;	//Disable digi. NCK input 38
   A_Disabl_Inp39 : BOOL ;	//Disable digi. NCK input 39
   A_Disabl_Inp40 : BOOL ;	//Disable digi. NCK input 40
   A_Set_Inp33 : BOOL ;	//Set digi. NCK input 33
   A_Set_Inp34 : BOOL ;	//Set digi. NCK input 34
   A_Set_Inp35 : BOOL ;	//Set digi. NCK input 35
   A_Set_Inp36 : BOOL ;	//Set digi. NCK input 36
   A_Set_Inp37 : BOOL ;	//Set digi. NCK input 37
   A_Set_Inp38 : BOOL ;	//Set digi. NCK input 38
   A_Set_Inp39 : BOOL ;	//Set digi. NCK input 39
   A_Set_Inp40 : BOOL ;	//Set digi. NCK input 40
   A_Disabl_Out9 : BOOL ;	//Disable digi. NCK output 9
   A_Disabl_Out10 : BOOL ;	//Disable digi. NCK output 10
   A_Disabl_Out11 : BOOL ;	//Disable digi. NCK output 11
   A_Disabl_Out12 : BOOL ;	//Disable digi. NCK output 12
   A_Disabl_Out13 : BOOL ;	//Disable digi. NCK output 13
   A_Disabl_Out14 : BOOL ;	//Disable digi. NCK output 14
   A_Disabl_Out15 : BOOL ;	//Disable digi. NCK output 15
   A_Disabl_Out16 : BOOL ;	//Disable digi. NCK output 16
   A_OvMask_Out9 : BOOL ;	//Overwrite mask of digi. output 9
   A_OvMask_Out10 : BOOL ;	//Overwrite mask of digi. output 10
   A_OvMask_Out11 : BOOL ;	//Overwrite mask of digi. output 11
   A_OvMask_Out12 : BOOL ;	//Overwrite mask of digi. output 12
   A_OvMask_Out13 : BOOL ;	//Overwrite mask of digi. output 13
   A_OvMask_Out14 : BOOL ;	//Overwrite mask of digi. output 14
   A_OvMask_Out15 : BOOL ;	//Overwrite mask of digi. output 15
   A_OvMask_Out16 : BOOL ;	//Overwrite mask of digi. output 16
   A_Setval_Out9 : BOOL ;	//Set value digi. NCK output 9
   A_Setval_Out10 : BOOL ;	//Set value digi. NCK output 10
   A_Setval_Out11 : BOOL ;	//Set value digi. NCK output 11
   A_Setval_Out12 : BOOL ;	//Set value digi. NCK output 12
   A_Setval_Out13 : BOOL ;	//Set value digi. NCK output 13
   A_Setval_Out14 : BOOL ;	//Set value digi. NCK output 14
   A_Setval_Out15 : BOOL ;	//Set value digi. NCK output 15
   A_Setval_Out16 : BOOL ;	//Set value digi. NCK output 16
   A_InMask_Out9 : BOOL ;	//Input mask of digi. output 9
   A_InMask_Out10 : BOOL ;	//Input mask of digi. output 10
   A_InMask_Out11 : BOOL ;	//Input mask of digi. output 11
   A_InMask_Out12 : BOOL ;	//Input mask of digi. output 12
   A_InMask_Out13 : BOOL ;	//Input mask of digi. output 13
   A_InMask_Out14 : BOOL ;	//Input mask of digi. output 14
   A_InMask_Out15 : BOOL ;	//Input mask of digi. output 15
   A_InMask_Out16 : BOOL ;	//Input mask of digi. output 16
   A_Disabl_Out17 : BOOL ;	//Disable digi. NCK output 17
   A_Disabl_Out18 : BOOL ;	//Disable digi. NCK output 18
   A_Disabl_Out19 : BOOL ;	//Disable digi. NCK output 19
   A_Disabl_Out20 : BOOL ;	//Disable digi. NCK output 20
   A_Disabl_Out21 : BOOL ;	//Disable digi. NCK output 21
   A_Disabl_Out22 : BOOL ;	//Disable digi. NCK output 22
   A_Disabl_Out23 : BOOL ;	//Disable digi. NCK output 23
   A_Disabl_Out24 : BOOL ;	//Disable digi. NCK output 24
   A_OvMask_Out17 : BOOL ;	//Overwrite mask of digi. output 17
   A_OvMask_Out18 : BOOL ;	//Overwrite mask of digi. output 18
   A_OvMask_Out19 : BOOL ;	//Overwrite mask of digi. output 19
   A_OvMask_Out20 : BOOL ;	//Overwrite mask of digi. output 20
   A_OvMask_Out21 : BOOL ;	//Overwrite mask of digi. output 21
   A_OvMask_Out22 : BOOL ;	//Overwrite mask of digi. output 22
   A_OvMask_Out23 : BOOL ;	//Overwrite mask of digi. output 23
   A_OvMask_Out24 : BOOL ;	//Overwrite mask of digi. output 24
   A_Setval_Out17 : BOOL ;	//Set value digi. NCK output 17
   A_Setval_Out18 : BOOL ;	//Set value digi. NCK output 18
   A_Setval_Out19 : BOOL ;	//Set value digi. NCK output 19
   A_Setval_Out20 : BOOL ;	//Set value digi. NCK output 20
   A_Setval_Out21 : BOOL ;	//Set value digi. NCK output 21
   A_Setval_Out22 : BOOL ;	//Set value digi. NCK output 22
   A_Setval_Out23 : BOOL ;	//Set value digi. NCK output 23
   A_Setval_Out24 : BOOL ;	//Set value digi. NCK output 24
   A_InMask_Out17 : BOOL ;	//Input mask of digi. output 17
   A_InMask_Out18 : BOOL ;	//Input mask of digi. output 18
   A_InMask_Out19 : BOOL ;	//Input mask of digi. output 19
   A_InMask_Out20 : BOOL ;	//Input mask of digi. output 20
   A_InMask_Out21 : BOOL ;	//Input mask of digi. output 21
   A_InMask_Out22 : BOOL ;	//Input mask of digi. output 22
   A_InMask_Out23 : BOOL ;	//Input mask of digi. output 23
   A_InMask_Out24 : BOOL ;	//Input mask of digi. output 24
   A_Disabl_Out25 : BOOL ;	//Disable digi. NCK output 25
   A_Disabl_Out26 : BOOL ;	//Disable digi. NCK output 26
   A_Disabl_Out27 : BOOL ;	//Disable digi. NCK output 27
   A_Disabl_Out28 : BOOL ;	//Disable digi. NCK output 28
   A_Disabl_Out29 : BOOL ;	//Disable digi. NCK output 29
   A_Disabl_Out30 : BOOL ;	//Disable digi. NCK output 30
   A_Disabl_Out31 : BOOL ;	//Disable digi. NCK output 31
   A_Disabl_Out32 : BOOL ;	//Disable digi. NCK output 32
   A_OvMask_Out25 : BOOL ;	//Overwrite mask of digi. output 25
   A_OvMask_Out26 : BOOL ;	//Overwrite mask of digi. output 26
   A_OvMask_Out27 : BOOL ;	//Overwrite mask of digi. output 27
   A_OvMask_Out28 : BOOL ;	//Overwrite mask of digi. output 28
   A_OvMask_Out29 : BOOL ;	//Overwrite mask of digi. output 29
   A_OvMask_Out30 : BOOL ;	//Overwrite mask of digi. output 30
   A_OvMask_Out31 : BOOL ;	//Overwrite mask of digi. output 31
   A_OvMask_Out32 : BOOL ;	//Overwrite mask of digi. output 32
   A_Setval_Out25 : BOOL ;	//Set value digi. NCK output 25
   A_Setval_Out26 : BOOL ;	//Set value digi. NCK output 26
   A_Setval_Out27 : BOOL ;	//Set value digi. NCK output 27
   A_Setval_Out28 : BOOL ;	//Set value digi. NCK output 28
   A_Setval_Out29 : BOOL ;	//Set value digi. NCK output 29
   A_Setval_Out30 : BOOL ;	//Set value digi. NCK output 30
   A_Setval_Out31 : BOOL ;	//Set value digi. NCK output 31
   A_Setval_Out32 : BOOL ;	//Set value digi. NCK output 32
   A_InMask_Out25 : BOOL ;	//Input mask of digi. output 25
   A_InMask_Out26 : BOOL ;	//Input mask of digi. output 26
   A_InMask_Out27 : BOOL ;	//Input mask of digi. output 27
   A_InMask_Out28 : BOOL ;	//Input mask of digi. output 28
   A_InMask_Out29 : BOOL ;	//Input mask of digi. output 29
   A_InMask_Out30 : BOOL ;	//Input mask of digi. output 30
   A_InMask_Out31 : BOOL ;	//Input mask of digi. output 31
   A_InMask_Out32 : BOOL ;	//Input mask of digi. output 32
   A_Disabl_Out33 : BOOL ;	//Disable digi. NCK output 33
   A_Disabl_Out34 : BOOL ;	//Disable digi. NCK output 34
   A_Disabl_Out35 : BOOL ;	//Disable digi. NCK output 35
   A_Disabl_Out36 : BOOL ;	//Disable digi. NCK output 36
   A_Disabl_Out37 : BOOL ;	//Disable digi. NCK output 37
   A_Disabl_Out38 : BOOL ;	//Disable digi. NCK output 38
   A_Disabl_Out39 : BOOL ;	//Disable digi. NCK output 39
   A_Disabl_Out40 : BOOL ;	//Disable digi. NCK output 40
   A_OvMask_Out33 : BOOL ;	//Overwrite mask of digi. output 33
   A_OvMask_Out34 : BOOL ;	//Overwrite mask of digi. output 34
   A_OvMask_Out35 : BOOL ;	//Overwrite mask of digi. output 35
   A_OvMask_Out36 : BOOL ;	//Overwrite mask of digi. output 36
   A_OvMask_Out37 : BOOL ;	//Overwrite mask of digi. output 37
   A_OvMask_Out38 : BOOL ;	//Overwrite mask of digi. output 38
   A_OvMask_Out39 : BOOL ;	//Overwrite mask of digi. output 39
   A_OvMask_Out40 : BOOL ;	//Overwrite mask of digi. output 40
   A_Setval_out33 : BOOL ;	//Set value digi. NCK output 33
   A_Setval_out34 : BOOL ;	//Set value digi. NCK output 34
   A_Setval_out35 : BOOL ;	//Set value digi. NCK output 35
   A_Setval_out36 : BOOL ;	//Set value digi. NCK output 36
   A_Setval_out37 : BOOL ;	//Set value digi. NCK output 37
   A_Setval_out38 : BOOL ;	//Set value digi. NCK output 38
   A_Setval_out39 : BOOL ;	//Set value digi. NCK output 39
   A_Setval_out40 : BOOL ;	//Set value digi. NCK output 40
   A_InMask_Out33 : BOOL ;	//Input mask of digi. output 33
   A_InMask_Out34 : BOOL ;	//Input mask of digi. output 34
   A_InMask_Out35 : BOOL ;	//Input mask of digi. output 35
   A_InMask_Out36 : BOOL ;	//Input mask of digi. output 36
   A_InMask_Out37 : BOOL ;	//Input mask of digi. output 37
   A_InMask_Out38 : BOOL ;	//Input mask of digi. output 38
   A_InMask_Out39 : BOOL ;	//Input mask of digi. output 39
   A_InMask_Out40 : BOOL ;	//Input mask of digi. output 40
   A_Disabl_anaIn1 : BOOL ;	//Disable analog NCK input 1
   A_Disabl_anaIn2 : BOOL ;	//Disable analog NCK input 2
   A_Disabl_anaIn3 : BOOL ;	//Disable analog NCK input 3
   A_Disabl_anaIn4 : BOOL ;	//Disable analog NCK input 4
   A_Disabl_anaIn5 : BOOL ;	//Disable analog NCK input 5
   A_Disabl_anaIn6 : BOOL ;	//Disable analog NCK input 6
   A_Disabl_anaIn7 : BOOL ;	//Disable analog NCK input 7
   A_Disabl_anaIn8 : BOOL ;	//Disable analog NCK input 8
   A_InMask_anaIn1 : BOOL ;	//Input mask of analog NCK input 1
   A_InMask_anaIn2 : BOOL ;	//Input mask of analog NCK input 2
   A_InMask_anaIn3 : BOOL ;	//Input mask of analog NCK input 3
   A_InMask_anaIn4 : BOOL ;	//Input mask of analog NCK input 4
   A_InMask_anaIn5 : BOOL ;	//Input mask of analog NCK input 5
   A_InMask_anaIn6 : BOOL ;	//Input mask of analog NCK input 6
   A_InMask_anaIn7 : BOOL ;	//Input mask of analog NCK input 7
   A_InMask_anaIn8 : BOOL ;	//Input mask of analog NCK input 8
   A_Setval_anaIn1 : WORD ;	//Set value of analog NCK input 1
   A_Setval_anaIn2 : WORD ;	//Set value of analog NCK input 2
   A_Setval_anaIn3 : WORD ;	//Set value of analog NCK input 3
   A_Setval_anaIn4 : WORD ;	//Set value of analog NCK input 4
   A_Setval_anaIn5 : WORD ;	//Set value of analog NCK input 5
   A_Setval_anaIn6 : WORD ;	//Set value of analog NCK input 6
   A_Setval_anaIn7 : WORD ;	//Set value of analog NCK input 7
   A_Setval_anaIn8 : WORD ;	//Set value of analog NCK input 8
   f164_f165 : INT ;
   A_OvMask_anaOut1 : BOOL ;	//Overwrite mask of analog output 1
   A_OvMask_anaOut2 : BOOL ;	//Overwrite mask of analog output 2
   A_OvMask_anaOut3 : BOOL ;	//Overwrite mask of analog output 3
   A_OvMask_anaOut4 : BOOL ;	//Overwrite mask of analog output 4
   A_OvMask_anaOut5 : BOOL ;	//Overwrite mask of analog output 5
   A_OvMask_anaOut6 : BOOL ;	//Overwrite mask of analog output 6
   A_OvMask_anaOut7 : BOOL ;	//Overwrite mask of analog output 7
   A_OvMask_anaOut8 : BOOL ;	//Overwrite mask of analog output 8
   A_InMask_anaOut1 : BOOL ;	//Input mask of analog NCK output 1
   A_InMask_anaOut2 : BOOL ;	//Input mask of analog NCK output 2
   A_InMask_anaOut3 : BOOL ;	//Input mask of analog NCK output 3
   A_InMask_anaOut4 : BOOL ;	//Input mask of analog NCK output 4
   A_InMask_anaOut5 : BOOL ;	//Input mask of analog NCK output 5
   A_InMask_anaOut6 : BOOL ;	//Input mask of analog NCK output 6
   A_InMask_anaOut7 : BOOL ;	//Input mask of analog NCK output 7
   A_InMask_anaOut8 : BOOL ;	//Input mask of analog NCK output 8
   A_Disabl_anaOut1 : BOOL ;	//Disable analog NCK output 1
   A_Disabl_anaOut2 : BOOL ;	//Disable analog NCK output 2
   A_Disabl_anaOut3 : BOOL ;	//Disable analog NCK output 3
   A_Disabl_anaOut4 : BOOL ;	//Disable analog NCK output 4
   A_Disabl_anaOut5 : BOOL ;	//Disable analog NCK output 5
   A_Disabl_anaOut6 : BOOL ;	//Disable analog NCK output 6
   A_Disabl_anaOut7 : BOOL ;	//Disable analog NCK output 7
   A_Disabl_anaOut8 : BOOL ;	//Disable analog NCK output 8
   f169 : BYTE ;
   A_Setval_anaOut1 : WORD ;	//Set value of analog NCK output 1
   A_Setval_anaOut2 : WORD ;	//Set value of analog NCK output 2
   A_Setval_anaOut3 : WORD ;	//Set value of analog NCK output 3
   A_Setval_anaOut4 : WORD ;	//Set value of analog NCK output 4
   A_Setval_anaOut5 : WORD ;	//Set value of analog NCK output 5
   A_Setval_anaOut6 : WORD ;	//Set value of analog NCK output 6
   A_Setval_anaOut7 : WORD ;	//Set value of analog NCK output 7
   A_Setval_anaOut8 : WORD ;	//Set value of analog NCK output 8
   E_ActVal_In9 : BOOL ;	//Actual value of digi. NCK input 9
   E_ActVal_In10 : BOOL ;	//Actual value of digi. NCK input 10
   E_ActVal_In11 : BOOL ;	//Actual value of digi. NCK input 11
   E_ActVal_In12 : BOOL ;	//Actual value of digi. NCK input 12
   E_ActVal_In13 : BOOL ;	//Actual value of digi. NCK input 13
   E_ActVal_In14 : BOOL ;	//Actual value of digi. NCK input 14
   E_ActVal_In15 : BOOL ;	//Actual value of digi. NCK input 15
   E_ActVal_In16 : BOOL ;	//Actual value of digi. NCK input 16
   E_ActVal_In17 : BOOL ;	//Actual value of digi. NCK input 17
   E_ActVal_In18 : BOOL ;	//Actual value of digi. NCK input 18
   E_ActVal_In19 : BOOL ;	//Actual value of digi. NCK input 19
   E_ActVal_In20 : BOOL ;	//Actual value of digi. NCK input 20
   E_ActVal_In21 : BOOL ;	//Actual value of digi. NCK input 21
   E_ActVal_In22 : BOOL ;	//Actual value of digi. NCK input 22
   E_ActVal_In23 : BOOL ;	//Actual value of digi. NCK input 23
   E_ActVal_In24 : BOOL ;	//Actual value of digi. NCK input 24
   E_ActVal_In25 : BOOL ;	//Actual value of digi. NCK input 25
   E_ActVal_In26 : BOOL ;	//Actual value of digi. NCK input 26
   E_ActVal_In27 : BOOL ;	//Actual value of digi. NCK input 27
   E_ActVal_In28 : BOOL ;	//Actual value of digi. NCK input 28
   E_ActVal_In29 : BOOL ;	//Actual value of digi. NCK input 29
   E_ActVal_In30 : BOOL ;	//Actual value of digi. NCK input 30
   E_ActVal_In31 : BOOL ;	//Actual value of digi. NCK input 31
   E_ActVal_In32 : BOOL ;	//Actual value of digi. NCK input 32
   E_ActVal_In33 : BOOL ;	//Actual value of digi. NCK input 33
   E_ActVal_In34 : BOOL ;	//Actual value of digi. NCK input 34
   E_ActVal_In35 : BOOL ;	//Actual value of digi. NCK input 35
   E_ActVal_In36 : BOOL ;	//Actual value of digi. NCK input 36
   E_ActVal_In37 : BOOL ;	//Actual value of digi. NCK input 37
   E_ActVal_In38 : BOOL ;	//Actual value of digi. NCK input 38
   E_ActVal_In39 : BOOL ;	//Actual value of digi. NCK input 39
   E_ActVal_In40 : BOOL ;	//Actual value of digi. NCK input 40
   E_Setpoint_Out9 : BOOL ;	//Setpoint of digi. NCK output 9
   E_Setpoint_Out10 : BOOL ;	//Setpoint of digi. NCK output 10
   E_Setpoint_Out11 : BOOL ;	//Setpoint of digi. NCK output 11
   E_Setpoint_Out12 : BOOL ;	//Setpoint of digi. NCK output 12
   E_Setpoint_Out13 : BOOL ;	//Setpoint of digi. NCK output 13
   E_Setpoint_Out14 : BOOL ;	//Setpoint of digi. NCK output 14
   E_Setpoint_Out15 : BOOL ;	//Setpoint of digi. NCK output 15
   E_Setpoint_Out16 : BOOL ;	//Setpoint of digi. NCK output 16
   E_Setpoint_Out17 : BOOL ;	//Setpoint of digi. NCK output 17
   E_Setpoint_Out18 : BOOL ;	//Setpoint of digi. NCK output 18
   E_Setpoint_Out19 : BOOL ;	//Setpoint of digi. NCK output 19
   E_Setpoint_Out20 : BOOL ;	//Setpoint of digi. NCK output 20
   E_Setpoint_Out21 : BOOL ;	//Setpoint of digi. NCK output 21
   E_Setpoint_Out22 : BOOL ;	//Setpoint of digi. NCK output 22
   E_Setpoint_Out23 : BOOL ;	//Setpoint of digi. NCK output 23
   E_Setpoint_Out24 : BOOL ;	//Setpoint of digi. NCK output 24
   E_Setpoint_Out25 : BOOL ;	//Setpoint of digi. NCK output 25
   E_Setpoint_Out26 : BOOL ;	//Setpoint of digi. NCK output 26
   E_Setpoint_Out27 : BOOL ;	//Setpoint of digi. NCK output 27
   E_Setpoint_Out28 : BOOL ;	//Setpoint of digi. NCK output 28
   E_Setpoint_Out29 : BOOL ;	//Setpoint of digi. NCK output 29
   E_Setpoint_Out30 : BOOL ;	//Setpoint of digi. NCK output 30
   E_Setpoint_Out31 : BOOL ;	//Setpoint of digi. NCK output 31
   E_Setpoint_Out32 : BOOL ;	//Setpoint of digi. NCK output 32
   E_Setpoint_Out33 : BOOL ;	//Setpoint of digi. NCK output 33
   E_Setpoint_Out34 : BOOL ;	//Setpoint of digi. NCK output 34
   E_Setpoint_Out35 : BOOL ;	//Setpoint of digi. NCK output 35
   E_Setpoint_Out36 : BOOL ;	//Setpoint of digi. NCK output 36
   E_Setpoint_Out37 : BOOL ;	//Setpoint of digi. NCK output 37
   E_Setpoint_Out38 : BOOL ;	//Setpoint of digi. NCK output 38
   E_Setpoint_Out39 : BOOL ;	//Setpoint of digi. NCK output 39
   E_Setpoint_Out40 : BOOL ;	//Setpoint of digi. NCK output 40
   E_ActVal_anaIn1 : WORD ;	//Actual value of analog NCK input 1
   E_ActVal_anaIn2 : WORD ;	//Actual value of analog NCK input 2
   E_ActVal_anaIn3 : WORD ;	//Actual value of analog NCK input 3
   E_ActVal_anaIn4 : WORD ;	//Actual value of analog NCK input 4
   E_ActVal_anaIn5 : WORD ;	//Actual value of analog NCK input 5
   E_ActVal_anaIn6 : WORD ;	//Actual value of analog NCK input 6
   E_ActVal_anaIn7 : WORD ;	//Actual value of analog NCK input 7
   E_ActVal_anaIn8 : WORD ;	//Actual value of analog NCK input 8
   E_SetVal_anaOut1 : WORD ;	//Set value of analog NCK output 1
   E_SetVal_anaOut2 : WORD ;	//Set value of analog NCK output 2
   E_SetVal_anaOut3 : WORD ;	//Set value of analog NCK output 3
   E_SetVal_anaOut4 : WORD ;	//Set value of analog NCK output 4
   E_SetVal_anaOut5 : WORD ;	//Set value of analog NCK output 5
   E_SetVal_anaOut6 : WORD ;	//Set value of analog NCK output 6
   E_SetVal_anaOut7 : WORD ;	//Set value of analog NCK output 7
   E_SetVal_anaOut8 : WORD ;	//Set value of analog NCK output 8
   E_CollCheck : ARRAY  [0 .. 7 ] OF BYTE ;	//CollisionsCheck
   A_CollCheck : ARRAY  [0 .. 7 ] OF BYTE ;	//CollisionsCheck
   E_HW4_moved : BYTE ;	//Handwheel 4 moved
   E_HW5_moved : BYTE ;	//Handwheel 5 moved
   E_HW6_moved : BYTE ;	//Handwheel 6 moved
   E_EHW1_stands : BOOL ;	//Ethernet handwheel 1 stands
   E_EHW2_stands : BOOL ;	//Ethernet handwheel 2 stands
   E_EHW3_stands : BOOL ;	//Ethernet handwheel 3 stands
   E_EHW4_stands : BOOL ;	//Ethernet handwheel 4 stands
   E_EHW5_stands : BOOL ;	//Ethernet handwheel 5 stands
   E_EHW6_stands : BOOL ;	//Ethernet handwheel 6 stands
   f245_6 : BOOL ;
   f245_7 : BOOL ;
   f246 : WORD ;
  END_STRUCT ;	
END_TYPE

TYPE UDT 11
VERSION : 0.0
  STRUCT
   A_AUTO : BOOL ;	//AUTOMATIC mode
   A_MDA : BOOL ;	//MDA mode
   A_JOG : BOOL ;	//JOG mode
   f0_3 : BOOL ;
   A_MCDisable : BOOL ;	//Mode change disable
   A_MGStop : BOOL ;	//Mode group stop
   A_MGStopASp : BOOL ;	//Mode group stop axes plus spindle
   A_MGReset : BOOL ;	//Mode group reset
   A_TEACHIN : BOOL ;	//Machine function TEACH IN
   A_REPOS : BOOL ;	//Machine function REPOS
   A_REF : BOOL ;	//Machine function REF
   f1_3 : BOOL ;
   f1_4 : BOOL ;
   f1_5 : BOOL ;
   A_SingleBlock_B : BOOL ;	// Single block type B
   A_SingleBlock_A : BOOL ;	// Single block type A
   A_INC1 : BOOL ;	//INC1
   A_INC10 : BOOL ;	//INC10
   A_INC100 : BOOL ;	//INC100
   A_INC1000 : BOOL ;	//INC1000
   A_INC10000 : BOOL ;	//INC10000
   A_INCVar : BOOL ;	//INC variable
   f3 : BYTE ;
   E_MMC_AUTO : BOOL ;	//MMC Strobe AUTOMATIC mode
   E_MMC_MDA : BOOL ;	//MMC Strobe MDA mode
   E_MMC_JOG : BOOL ;	//MMC Strobe JOG mode
   f4_3 : BOOL ;
   f4_4 : BOOL ;
   f4_5 : BOOL ;
   f4_6 : BOOL ;
   f4_7 : BOOL ;
   E_MMC_TEACHIN : BOOL ;	//MMC Strobe machine function TEACH IN
   E_MMC_REPOS : BOOL ;	//MMC Strobe machine function REPOS
   E_MMC_REF : BOOL ;	//MMC Strobe Machine function REF
   f5_3 : BOOL ;
   f5_4 : BOOL ;
   f5_5 : BOOL ;
   f5_6 : BOOL ;
   f5_7 : BOOL ;
   E_AUTO : BOOL ;	//Active AUTOMATIC mode
   E_MDA : BOOL ;	//Active MDA mode
   E_JOG : BOOL ;	//Active JOG mode
   E_MGOK : BOOL ;	//Mode group ready
   E_MGreseted : BOOL ;	// Mode Group reseted
   E_NCKintJOG : BOOL ;	// NCK internal JOG active
   f6_6 : BOOL ;
   E_ChanReset : BOOL ;	//All channels in reset state
   E_TEACHIN : BOOL ;	//Active machine function TEACH IN
   E_REPOS : BOOL ;	//Active machine function REPOS
   E_REF : BOOL ;	//Active Machine function REF
   f7_3 : BOOL ;
   f7_4 : BOOL ;
   f7_5 : BOOL ;
   f7_6 : BOOL ;
   f7_7 : BOOL ;
   E_INC1 : BOOL ;	//INC1
   E_INC10 : BOOL ;	//INC10
   E_INC100 : BOOL ;	//INC100
   E_INC1000 : BOOL ;	//INC1000
   E_INC10000 : BOOL ;	//INC10000
   E_INCVar : BOOL ;	//INC variable
   f8_6 : BOOL ;
   f8_7 : BOOL ;
   f9 : BYTE ;
   f10 : ARRAY  [10 .. 19 ] OF BYTE ;
   MG : ARRAY  [2 .. 10 ] OF STRUCT
    A_AUTO : BOOL ;	//AUTOMATIC mode
    A_MDA : BOOL ;	//MDA mode
    A_JOG : BOOL ;	//JOG mode
    f0_3 : BOOL ;
    A_MCDisable : BOOL ;	//Mode change disable
    A_MGStop : BOOL ;	//Mode group stop
    A_MGStopASp : BOOL ;	//Mode group stop axes plus spindle
    A_MGReset : BOOL ;	//Mode group reset
    A_TEACHIN : BOOL ;	//Machine function TEACH IN
    A_REPOS : BOOL ;	//Machine function REPOS
    A_REF : BOOL ;	//Machine function REF
    f1_3 : BOOL ;
    f1_4 : BOOL ;
    f1_5 : BOOL ;
    A_SingleBlock_B : BOOL ;	// Single block type B
    A_SingleBlock_A : BOOL ;	// Single block type A
    A_INC1 : BOOL ;	//INC1
    A_INC10 : BOOL ;	//INC10
    A_INC100 : BOOL ;	//INC100
    A_INC1000 : BOOL ;	//INC1000
    A_INC10000 : BOOL ;	//INC10000
    A_INCVar : BOOL ;	//INC variable
    f3 : BYTE ;
    E_MMC_AUTO : BOOL ;	//MMC Strobe AUTOMATIC mode
    E_MMC_MDA : BOOL ;	//MMC Strobe MDA mode
    E_MMC_JOG : BOOL ;	//MMC Strobe JOG mode
    f4_3 : BOOL ;
    f4_4 : BOOL ;
    f4_5 : BOOL ;
    f4_6 : BOOL ;
    f4_7 : BOOL ;
    E_MMC_TEACHIN : BOOL ;	//MMC Strobe machine function TEACH IN
    E_MMC_REPOS : BOOL ;	//MMC Strobe machine function REPOS
    E_MMC_REF : BOOL ;	//MMC Strobe Machine function REF
    f5_3 : BOOL ;
    f5_4 : BOOL ;
    f5_5 : BOOL ;
    f5_6 : BOOL ;
    f5_7 : BOOL ;
    E_AUTO : BOOL ;	//Active AUTOMATIC mode
    E_MDA : BOOL ;	//Active MDA mode
    E_JOG : BOOL ;	//Active JOG mode
    E_MGOK : BOOL ;	//Mode group ready
    E_MGreseted : BOOL ;	// Mode Group reseted
    E_NCKintJOG : BOOL ;	// NCK internal JOG active
    f6_6 : BOOL ;
    E_ChanReset : BOOL ;	//All channels in reset state
    E_TEACHIN : BOOL ;	//Active machine function TEACH IN
    E_REPOS : BOOL ;	//Active machine function REPOS
    E_REF : BOOL ;	//Active machine function REF
    f7_3 : BOOL ;
    f7_4 : BOOL ;
    f7_5 : BOOL ;
    f7_6 : BOOL ;
    f7_7 : BOOL ;
    E_INC1 : BOOL ;	//INC1
    E_INC10 : BOOL ;	//INC10
    E_INC100 : BOOL ;	//INC100
    E_INC1000 : BOOL ;	//INC1000
    E_INC10000 : BOOL ;	//INC10000
    E_INCVar : BOOL ;	//INC variable
    f8_6 : BOOL ;
    f8_7 : BOOL ;
    f9 : BYTE ;
    f10 : ARRAY  [10 .. 19 ] OF BYTE ;
   END_STRUCT ;
  END_STRUCT ;	
END_TYPE

TYPE UDT 19
VERSION : 0.0
  STRUCT
   A_SCLight : BOOL ;	//Screen light
   A_SCDark : BOOL ;	//Screen darkening
   A_KeyDisable : BOOL ;	//Key disable
   A_ClearCanAl : BOOL ;	//Clear cancel alarms
   A_ClearRecAl : BOOL ;	//Clear recall alarms
   f0_5 : BOOL ;
   f0_6 : BOOL ;
   A_ActWCS : BOOL ;	//Actual value in WCS 0=MCS
   A_PLCExtViewerReject : BOOL ;	//External viewer reject
   A_PLCExtViewerMode : BOOL ;	//External viewer mode
   f1_2 : BOOL ;
   f1_3 : BOOL ;
   f1_4 : BOOL ;
   f1_5 : BOOL ;
   f1_6 : BOOL ;
   f1_7 : BOOL ;
   A_1stError1 : WORD ;	//1st error HIGRAPH
   A_1stError2 : WORD ;	//1st error HIGRAPH
   A_ASpi1percent : BYTE ;	//Analog spindle 1:
   A_ASpi2percent : BYTE ;
   A_MCPChan : BYTE ;
   A_OEM1 : BOOL ;
   A_OEM2 : BOOL ;
   A_AToolMeas : BOOL ;	//AutoToolMeasure
   f9_3 : BOOL ;
   f9_4 : BOOL ;
   f9_5 : BOOL ;
   f9_6 : BOOL ;
   f9_7 : BOOL ;
   A_Hardkey : BYTE ;	//PLC Hardkeys
   f11 : BYTE ;	//Reserved for hardkeys
   f12_0 : BOOL ;
   f12_1 : BOOL ;
   A_COM2 : BOOL ;
   A_COM1 : BOOL ;
   A_V24stop : BOOL ;
   A_V24ext : BOOL ;
   A_V24off : BOOL ;
   A_V24on : BOOL ;
   A_TeachDisable : BOOL ;
   f13_1 : BOOL ;
   f13_2 : BOOL ;
   f13_3 : BOOL ;
   f13_4 : BOOL ;
   A_PPdeload : BOOL ;
   A_PPload : BOOL ;
   A_PPsel : BOOL ;
   A_V24Index1 : BYTE ;
   A_V24Index2 : BYTE ;
   A_V24NoFile1 : BYTE ;
   A_V24NoFile2 : BYTE ;
   A_res18 : BYTE ;
   A_res19 : BYTE ;	//Message counter
   f20_0 : BOOL ;
   E_SCDark : BOOL ;	//Screen darkening
   E_Cancel : BOOL ;	//Cancel
   E_CanCleared : BOOL ;	//Cancel alarms cleared
   E_RecCleared : BOOL ;	//Recall alarms cleared
   f20_5 : BOOL ;	//res. Language
   E_SimActiv : BOOL ;	//Simulation active
   E_ActWCS : BOOL ;	//Switchover MCS/WCS 0=MCS
   E_ActivWA : BYTE ;
   E_Chan : BYTE ;	//Channel displayed
   E_KeybHandl : BOOL ;	// Keyboard handling
   E_DataTransf : BOOL ;	// Data transfer active
   E_DisplChange : BOOL ;	// Display change
   f23_3 : BOOL ;
   f23_4 : BOOL ;
   f23_5 : BOOL ;
   f23_6 : BOOL ;
   f23_7 : BOOL ;
   E_V24Err : BOOL ;
   E_V24OK : BOOL ;
   E_V24COM2 : BOOL ;
   E_V24COM1 : BOOL ;
   E_V24stop : BOOL ;
   E_V24ext : BOOL ;
   E_V24off : BOOL ;
   E_V24on : BOOL ;
   E_V24Error : BYTE ;	//V24: Error Byte
   E_res26_0 : BOOL ;	//Reserved
   E_PPOK : BOOL ;	//Part program status OK
   E_PPErr : BOOL ;	//Part program status Error
   E_PPAct : BOOL ;	//Part program status active
   f26_4 : BOOL ;	//Reserved
   E_PPdeload : BOOL ;	//Part program status deloading
   E_PPload : BOOL ;	//Part program status loading
   E_PPsel : BOOL ;	//Part program status selecting
   E_PPError : BYTE ;	//Part program status Error
   A_PictNo : INT ;
   A_PictOn : BOOL ;
   A_PictOff : BOOL ;
   f30_2 : BOOL ;
   f30_3 : BOOL ;
   f30_4 : BOOL ;
   f30_5 : BOOL ;
   f30_6 : BOOL ;
   f30_7 : BOOL ;
   E_PictOK : BOOL ;
   E_PictOn : BOOL ;
   E_PictAct : BOOL ;
   E_PictOff : BOOL ;
   E_PictErr : BOOL ;
   f31_5 : BOOL ;
   f31_6 : BOOL ;
   E_NotAct : BOOL ;
   A_FuncNo : BYTE ;
   A_Par1 : BYTE ;
   A_Par2 : BYTE ;
   A_Par3 : BYTE ;
   E_FuncErr : BYTE ;
   f37 : BYTE ;
   f38 : BYTE ;
   f39 : BYTE ;
   res40 : ARRAY  [0 .. 9 ] OF BYTE ;
   MMC2 : STRUCT
    A_SCLight : BOOL ;	//Screen light
    A_SCDark : BOOL ;	//Screen darkening
    A_KeyDisable : BOOL ;	//Key disable
    A_ClearCanAl : BOOL ;	//Clear cancel alarms
    A_ClearRecAl : BOOL ;	//Clear recall alarms
    f0_5 : BOOL ;
    f0_6 : BOOL ;
    A_ActWCS : BOOL ;	//Actual value in WCS 0=MCS
    A_1stError1 : WORD ;	//1st error HIGRAPH
    A_1stError2 : WORD ;	//1st error HIGRAPH
    A_ASpi1percent : BYTE ;	//Analog spindle 1:
    A_ASpi2percent : BYTE ;
    A_MCPChan : BYTE ;
    A_OEM1 : BOOL ;
    A_OEM2 : BOOL ;
    A_AToolMeas : BOOL ;	//AutoToolMeasure
    f9_3 : BOOL ;
    f9_4 : BOOL ;
    f9_5 : BOOL ;
    f9_6 : BOOL ;
    f9_7 : BOOL ;
    A_Hardkey : BYTE ;	//PLC Hardkeys
    f11 : BYTE ;	//Reserved for hardkeys
    f12_0 : BOOL ;
    f12_1 : BOOL ;
    A_COM2 : BOOL ;
    A_COM1 : BOOL ;
    A_V24stop : BOOL ;
    A_V24ext : BOOL ;
    A_V24off : BOOL ;
    A_V24on : BOOL ;
    f13_0 : BOOL ;
    f13_1 : BOOL ;
    f13_2 : BOOL ;
    f13_3 : BOOL ;
    f13_4 : BOOL ;
    A_PPdeload : BOOL ;
    A_PPload : BOOL ;
    A_PPsel : BOOL ;
    A_V24Index1 : BYTE ;
    A_V24Index2 : BYTE ;
    A_V24NoFile1 : BYTE ;
    A_V24NoFile2 : BYTE ;
    A_res18 : BYTE ;
    A_res19 : BYTE ;	//Message counter
    f20_0 : BOOL ;
    E_SCDark : BOOL ;	//Screen darkening
    E_Cancel : BOOL ;	//Cancel
    E_CanCleared : BOOL ;	//Cancel alarms cleared
    E_RecCleared : BOOL ;	//Recall alarms cleared
    f20_5 : BOOL ;	//res. Language
    E_SimActiv : BOOL ;	//Simulation active
    E_ActWCS : BOOL ;	//Switchover MCS/WCS 0=MCS
    E_ActivWA : BYTE ;
    E_Chan : BYTE ;	//Channel displayed
    f23 : BYTE ;
    E_V24Err : BOOL ;
    E_V24OK : BOOL ;
    E_V24COM2 : BOOL ;
    E_V24COM1 : BOOL ;
    E_V24stop : BOOL ;
    E_V24ext : BOOL ;
    E_V24off : BOOL ;
    E_V24on : BOOL ;
    E_V24Error : BYTE ;	//V24: Error Byte
    E_res26_0 : BOOL ;	//Reserved
    E_PPOK : BOOL ;	//Part program status OK
    E_PPErr : BOOL ;	//Part program status Error
    E_PPAct : BOOL ;	//Part program status active
    f26_4 : BOOL ;	//Reserved
    E_PPdeload : BOOL ;	//Part program status deloading
    E_PPload : BOOL ;	//Part program status loading
    E_PPsel : BOOL ;	//Part program status selecting
    E_PPError : BYTE ;	//Part program status Error
    A_PictNo : INT ;
    A_PictOn : BOOL ;
    A_PictOff : BOOL ;
    f30_2 : BOOL ;
    f30_3 : BOOL ;
    f30_4 : BOOL ;
    f30_5 : BOOL ;
    f30_6 : BOOL ;
    f30_7 : BOOL ;
    E_PictOK : BOOL ;
    E_PictOn : BOOL ;
    E_PictAct : BOOL ;
    E_PictOff : BOOL ;
    E_PictErr : BOOL ;
    f31_5 : BOOL ;
    f31_6 : BOOL ;
    E_NotAct : BOOL ;
    A_FuncNo : BYTE ;
    A_Par1 : BYTE ;
    A_Par2 : BYTE ;
    A_Par3 : BYTE ;
    E_FuncErr : BYTE ;
    f37 : BYTE ;
    f38 : BYTE ;
    f39 : BYTE ;
    res40 : ARRAY  [0 .. 9 ] OF BYTE ;
   END_STRUCT ;	//M to N
   ONL_REQUEST : WORD ;
   ONL_CONFIRM : WORD ;
   PAR_CLIENT_IDENT : WORD ;
   PAR_MMC_TYP : BYTE ;
   PAR_MSTT_ADR : BYTE ;
   PAR_STATUS : BYTE ;
   PAR_Z_INFO : BYTE ;
   MtoNAlive : WORD ;
   f112 : BYTE ;
   ParOpKeyAdr : BYTE ;
   ParTcuIndex : BYTE ;
   f115 : BYTE ;
   Tcu1KeyAdr : BYTE ;
   Tcu2KeyAdr : BYTE ;
   Tcu1Index : BYTE ;
   Tcu2Index : BYTE ;
   MMC1_CLIENT_IDENT : WORD ;
   MMC1_TYP : BYTE ;
   MMC1_MSTT_ADR : BYTE ;
   MMC1_STATUS : BYTE ;
   MMC1_Z_INFO : BYTE ;
   MMC1_SHIFT_LOCK : BOOL ;
   MMC1_MSTT_SHIFT_LOCK : BOOL ;
   MMC1_ACTIVE_REQ : BOOL ;
   MMC1_ACTIVE_PERM : BOOL ;
   MMC1_ACTIVE_CHANGED : BOOL ;
   MMC1_CHANGED_DENIED : BOOL ;
   MMC1_TCU_SHIFT_LOCK : BOOL ;
   f127 : BYTE ;
   MMC1_TRANS_DB : WORD ;
   MMC2_CLIENT_IDENT : WORD ;
   MMC2_TYP : BYTE ;
   MMC2_MSTT_ADR : BYTE ;
   MMC2_STATUS : BYTE ;
   MMC2_Z_INFO : BYTE ;
   MMC2_SHIFT_LOCK : BOOL ;
   MMC2_MSTT_SHIFT_LOCK : BOOL ;
   MMC2_ACTIVE_REQ : BOOL ;
   MMC2_ACTIVE_PERM : BOOL ;
   MMC2_ACTIVE_CHANGED : BOOL ;
   MMC2_CHANGED_DENIED : BOOL ;
   MMC2_TCU_SHIFT_LOCK : BOOL ;
   f137 : BYTE ;
   MMC2_TRANS_DB : WORD ;
   A_Subtype : INT ;	//for Codecarrier Input from PLC
   A_Duplo : INT ;
   A_Ident : STRING  [32 ];
   A_Tnumber : INT ;
   A_MagazinePlace : INT ;
   A_MagazinePlaceType : INT ;
   A_ToolSize_Upper : BYTE ;
   A_ToolSize_Down : BYTE ;
   A_ToolSize_Left : BYTE ;
   A_ToolSize_Right : BYTE ;
   A_Channel : BYTE ;
   A_LoadingPlace : BYTE ;
   A_Magazine : INT ;
   A_Unit : BYTE ;
   A_NCU_Index : BYTE ;
   A_FileIndex : INT ;
   A_ActiveEnable : BOOL ;
   A_Override : BOOL ;
   A_LoadTool : BOOL ;
   A_DeleteTool : BOOL ;
   E_Subtype : INT ;	//for Codecarrier Output to PLC
   E_Duplo : INT ;
   E_Ident : STRING  [32 ];
   E_Tnumber : INT ;
   E_ToolState : INT ;
   E_MagazinePlaceType : INT ;
   E_ToolSize_Upper : BYTE ;
   E_ToolSize_Down : BYTE ;
   E_ToolSize_Left : BYTE ;
   E_ToolSize_Right : BYTE ;
   E_Magazine : INT ;
   E_MagazinePlace : INT ;
   A_ReqMMC1 : BOOL ;	//for Codecarrier Request MMC-Interface1
   A_ReqMMC2 : BOOL ;	//for Codecarrier Request MMC-Interface2
   A_K_Code : BYTE ;
   E_Done : BOOL ;
   E_Error : BOOL ;
   E_Active : BOOL ;	// CodeCarrierReadEnable : BOOL;
// CodeCarrierWriteEnable : BOOL;
   E_K_CodeError : BYTE ;	//Identify for Error_Code
   E_Error_Code : INT ;
   E_Req : BOOL ;	//for Positioning
   f257 : BYTE ;
   A_Done : BOOL ;
   A_Error : BOOL ;
   A_Active : BOOL ;
   f258_3 : BOOL ;
   f258_4 : BOOL ;
   f258_5 : BOOL ;
   f258_6 : BOOL ;
   f258_7 : BOOL ;
   E_TDC_Read : BOOL ;
   E_TDC_Write : BOOL ;
   E_TDC_Cancel : BOOL ;
   A_Error_Code : INT ;
   E_PMagazine : INT ;
   E_PMagazinePlace : INT ;
   E_PTnumber : INT ;	//TPM-Data
   A_TPMStatus : INT ;
   A_TPMCounter : ARRAY  [1 .. 32 ] OF DINT ;
   A_HWeelSimOvr : BYTE ;
   f399 : BYTE ;
   A_SimOvr : INT ;	// simulation overide
   A_SimState : INT ;	// simulation state
  END_STRUCT ;	
END_TYPE

TYPE UDT 21
VERSION : 0.0
  STRUCT
   f0_0 : BOOL ;
   f0_1 : BOOL ;
   f0_2 : BOOL ;
   A_DRF : BOOL ;	//Activate DRF
   A_SBL : BOOL ;	//Activate single block
   A_M01 : BOOL ;	//Activate M01
   A_DRY : BOOL ;	//Activate dry run feedrate
   f0_7 : BOOL ;
   A_Ref : BOOL ;	//Activate referencing
   A_ProtZone : BOOL ;	//Enable protection zones
   A_SynOff : BOOL ;	//Synchronous action off
   A_TM_TimOut : BOOL ;	//Activate time-out (TM)
   A_CLC_Stop : BOOL ;	//CLC stop
   A_CLC_OR : BOOL ;	//CLC override
   A_PLC_ActCompl : BOOL ;	//PLC action complete
   A_ProgTest : BOOL ;	//Activate program test
   A_SKP0 : BOOL ;	//Activate skip block \0
   A_SKP1 : BOOL ;	//Activate skip block \1
   A_SKP2 : BOOL ;	//Activate skip block \2
   A_SKP3 : BOOL ;	//Activate skip block \3
   A_SKP4 : BOOL ;	//Activate skip block \4
   A_SKP5 : BOOL ;	//Activate skip block \5
   A_SKP6 : BOOL ;	//Activate skip block \6
   A_SKP7 : BOOL ;	//Activate skip block \7
   A_StrokEnab : BOOL ;	//Stroke enable
   A_ManStrokEnab : BOOL ;	//Manual stroke enable
   A_StrokSup : BOOL ;	//Stroke suppression
   A_StrokDelayed : BOOL ;	//Stroke delayed
   A_StrokStop : BOOL ;	//Stroke not operating
   A_ManRelStroke2 : BOOL ;	// Manual release of stroke 2
   A3_6 : BOOL ;
   A3_7 : BOOL ;
   A_FD_OR : BYTE ;	//Feedrate override
   A_RT_OR : BYTE ;	//Rapid traverse override
   A_FDdisable : BOOL ;	//Feed disable
   A_RIdisable : BOOL ;	//Read-in disable
   A_DeleteDTG : BOOL ;	//Delete distance to go
   A_SP_Clear : BOOL ;	//Clear SP repetitions
   A_ProgAbort : BOOL ;	//Program level abort
   A_F_Limit : BOOL ;	//Tool path feedrate limitation
   A_RT_ORA : BOOL ;	//Rapid traverse override active
   A_FD_ORA : BOOL ;	//Feedrate override active
   A_NCStartDisabl : BOOL ;	//NC start disable
   A_NCStart : BOOL ;	//NC start
   A_NCStopBlock : BOOL ;	//NC stop at block limit
   A_NCStop : BOOL ;	//NC stop
   A_NCStopASp : BOOL ;	//NC stop axes plus spindle
   A_SuppStartLock : BOOL ;	// Suppress Start Lock
   f7_6 : BOOL ;
   A_Reset : BOOL ;	//Reset
   A_MRP : ARRAY  [1 .. 10 ] OF BOOL ;	//Activate machine-related protection area [1..10]
   A_CSP : ARRAY  [1 .. 10 ] OF BOOL ;	//Activate channel-specific protection area [1..10]
   A_Geo : ARRAY  [1 .. 3 ] OF STRUCT 	//Control signals for geometry axis [1..3]
    HW1 : BOOL ;	//Activate handwheel 1
    HW2 : BOOL ;	//Activate handwheel 2
    HW3 : BOOL ;	//Activate handwheel 3
    FDStop : BOOL ;	//Feed stop
    Disabl : BOOL ;	//Traversing key disable
    RapidTrOR : BOOL ;	//Rapid traverse override
    Minus : BOOL ;	//Traversing key minus
    Plus : BOOL ;	//Traversing key plus
    INC1 : BOOL ;	//INC 1
    INC10 : BOOL ;	//INC 10
    INC100 : BOOL ;	//INC 100
    INC1000 : BOOL ;	//INC 1000
    INC10000 : BOOL ;	//INC 10000
    INCVar : BOOL ;	//INC variable
    OEM : BYTE ;	//OEM signals
    InvHWDirOfRot : BOOL ;	// Inverting handwheel direction of rotation
    f3_1 : BOOL ;
    f3_2 : BOOL ;
    f3_3 : BOOL ;
    f3_4 : BOOL ;
    f3_5 : BOOL ;
    f3_6 : BOOL ;
    f3_7 : BOOL ;
   END_STRUCT ;
   f24_0 : BOOL ;
   f24_1 : BOOL ;
   f24_2 : BOOL ;
   E_MMC_DRF : BOOL ;	//MMC DRF selected
   f24_4 : BOOL ;
   E_MMC_M01 : BOOL ;	//MMC M01 selected
   E_MMC_DRY : BOOL ;	//MMC Dry run feedrate selected
   f24_7 : BOOL ;
   E_MMC_REPOSPM_0 : BOOL ;	//MMC REPOSPATHMODE 0
   E_MMC_REPOSPM_1 : BOOL ;	//MMC REPOSPATHMODE 1
   E_MMC_REPOSPM_2 : BOOL ;	//MMC REPOSPATHMODE 2
   E_MMC_FD_OR4RT_OR : BOOL ;	//MMC Feedrate override for rapid traverse selected
   E_MMC_REPOSMode : BOOL ;	//MMC REPOS MODE EDGE
   f25_5 : BOOL ;
   f25_6 : BOOL ;
   E_MMC_ProgTest : BOOL ;	//Program test selected
   E_MMC_SKP0 : BOOL ;	//MMC skip block selected \0
   E_MMC_SKP1 : BOOL ;	//MMC skip block selected \1
   E_MMC_SKP2 : BOOL ;	//MMC skip block selected \2
   E_MMC_SKP3 : BOOL ;	//MMC skip block selected \3
   E_MMC_SKP4 : BOOL ;	//MMC skip block selected \4
   E_MMC_SKP5 : BOOL ;	//MMC skip block selected \5
   E_MMC_SKP6 : BOOL ;	//MMC skip block selected \6
   E_MMC_SKP7 : BOOL ;	//MMC skip block selected \7
   E_MMC_SKP8 : BOOL ;	//MMC skip block selected \8
   E_MMC_SKP9 : BOOL ;	//MMC skip block selected \9
   f27_2 : BOOL ;
   f27_3 : BOOL ;
   f27_4 : BOOL ;
   f27_5 : BOOL ;
   f27_6 : BOOL ;
   f27_7 : BOOL ;
   A_OEM : BYTE ;
   A_FixedFD1 : BOOL ;	//Fixed feeds
   A_FixedFD2 : BOOL ;
   A_FixedFD3 : BOOL ;
   A_FixedFD4 : BOOL ;
   A_PTP_Travel : BOOL ;	//Activate PTP travel
   A_DisablWP_Counter : BOOL ;	//Disable workpiece counter
   A_DisablWearMon : BOOL ;	//Disable wear monitoring
   A_DontDisablTool : BOOL ;	//Do not disable tool
   A_ContHW1 : BOOL ;	//Activate contour handwheels
   A_ContHW2 : BOOL ;
   A_ContHW3 : BOOL ;
   A_ContHWsim : BOOL ;	//Simulated contour handwheel on
   A_ContHWneg : BOOL ;	//Contour handwheel neg. route
   A_NCKrelatedM01 : BOOL ;	// Activate NCK-related M01
   A_JOG_Circles : BOOL ;	// JOG in circles
   A_NoToolChangeCmd : BOOL ;	// No tool change commands
   A_REPOSPM_0 : BOOL ;	//REPOSPATHMODE 0
   A_REPOSPM_1 : BOOL ;	//REPOSPATHMODE 1
   A_REPOSPM_2 : BOOL ;	//REPOSPATHMODE 2
   f31_3 : BOOL ;
   A_REPOSMode : BOOL ;	//REPOS MODE EDGE
   A_InvCHWDirOfRot : BOOL ;	// Inverting contour handwheel direction of rotation
   A_SKP8 : BOOL ;	//Activate skip block \8
   A_SKP9 : BOOL ;	//Activate skip block \9
   E_ExecExtern : BOOL ;	//Execution from external source active
   f32_1 : BOOL ;
   f32_2 : BOOL ;
   E_ActBlock : BOOL ;	//Action block active
   E_BegBlock : BOOL ;	//Approach block active
   E_M01 : BOOL ;	//M0/M1 active
   E_LastActBlock : BOOL ;	//Last action block active
   f32_7 : BOOL ;
   E_Ref : BOOL ;	//Referencing active
   E_OrieToolholder : BOOL ;	// Orientable toolholder active
   E_RevFD : BOOL ;	//Revolutional feedrate active
   E_HWOverlay : BOOL ;	//Handwheel overlay active
   E_BlockSearch : BOOL ;	//Block search active
   E_M30 : BOOL ;	//M2/M30 active
   E_Transform : BOOL ;	//Transformation active
   E_ProgTest : BOOL ;	//Program test active
   E_OEMChan : BYTE ;	//OEM channel signals feedback
   E_ProgRunn : BOOL ;	//Program running
   E_ProgWait : BOOL ;	//Program waiting
   E_ProgStop : BOOL ;	//Program stopped
   E_ProgInterrupt : BOOL ;	//Program interrupted
   E_ProgrAborted : BOOL ;	//Program aborted
   E_ChanActive : BOOL ;	//Channel active
   E_ChanInterrupt : BOOL ;	//Channel interrupted
   E_ChanReset : BOOL ;	//Channel reset
   E_StartReq : BOOL ;	//Start request
   E_StopReq : BOOL ;	//Stop request
   E_AxesRef : BOOL ;	//All axes referenced
   E_AxesStop : BOOL ;	//All axes stationary
   E_IR_Activ : BOOL ;	//Interrupt processing active
   E_ChanRO : BOOL ;	//Channel ready for operation
   E_NCKalarmChan : BOOL ;	//Channel-specific NCK alarm present
   E_NCKalarmStop : BOOL ;	//NCK alarm with processing stop present
   E_CHW1 : BOOL ;	//Contour handwheel 1 on
   E_CHW2 : BOOL ;	//Contour handwheel 2 on
   E_CHW3 : BOOL ;	//Contour handwheel 3 on
   E_CLC : BOOL ;	//CLC active
   E_CLCStopLL : BOOL ;	//CLC stopped lower limit
   E_CLCStopUL : BOOL ;	//CLC stopped upper limit
   E_RIEnabIgnored : BOOL ;	//Read-in enable is ignored
   E_StopBlkEndSBLsuppr : BOOL ;	//Stop at block end with SBL is suppressed
   E_StrokeEA : BOOL ;	//Stroke enable active
   E_AcknManStrokEnab : BOOL ;	//Acknowledgement manual stroke enable
   f38_2 : BOOL ;
   f38_3 : BOOL ;
   f38_4 : BOOL ;
   f38_5 : BOOL ;
   f38_6 : BOOL ;
   f38_7 : BOOL ;
   E_ProtZoneNOK : BOOL ;	//Protection zones not guaranteed
   f39_1 : BOOL ;
   f39_2 : BOOL ;
   f39_3 : BOOL ;
   f39_4 : BOOL ;
   E_InvCHWDirOfRot : BOOL ;	// Contour handwheel direction of rotation invert actively
   f39_6 : BOOL ;
   f39_7 : BOOL ;
   E_Geo : ARRAY  [1 .. 3 ] OF STRUCT 	//Status signals of geometry axis [1..3]
    HW1 : BOOL ;	//Handwheel 1 active
    HW2 : BOOL ;	//Handwheel 2 active
    HW3 : BOOL ;	//Handwheel 3 active
    f0_3 : BOOL ;
    TReqMinus : BOOL ;	// Travel requests minus
    TReqPlus : BOOL ;	// Travel requests plus
    TCMinus : BOOL ;	//Traverse command minus
    TCPlus : BOOL ;	//Traverse command plus
    INC1 : BOOL ;	//INC 1 active
    INC10 : BOOL ;	//INC 10 active
    INC100 : BOOL ;	//INC 100 active
    INC1000 : BOOL ;	//INC 1000 active
    INC10000 : BOOL ;	//INC 10000 active
    INCVar : BOOL ;	//INC variable active
    OEM : BYTE ;	//OEM signals
    InvHWDirOfRot : BOOL ;	// Handwheel direction of rotation invert actively
    f3_1 : BOOL ;
    f3_2 : BOOL ;
    f3_3 : BOOL ;
    f3_4 : BOOL ;
    f3_5 : BOOL ;
    f3_6 : BOOL ;
    f3_7 : BOOL ;
    f4 : BYTE ;
   END_STRUCT ;
   M1Change : BOOL ;	//M function 1 change
   M2Change : BOOL ;	//M function 2 change
   M3Change : BOOL ;	//M function 3 change
   M4Change : BOOL ;	//M function 4 change
   M5Change : BOOL ;	//M function 5 change
   f58_5 : BOOL ;
   f58_6 : BOOL ;
   f58_7 : BOOL ;
   M1NDec : BOOL ;	//M function 1 not decoded
   M2NDec : BOOL ;	//M function 2 not decoded
   M3NDec : BOOL ;	//M function 3 not decoded
   M4NDec : BOOL ;	//M function 4 not decoded
   M5NDec : BOOL ;	//M function 5 not decoded
   f59_5 : BOOL ;
   f59_6 : BOOL ;
   f59_7 : BOOL ;
   S1Change : BOOL ;	//S function 1 change
   S2Change : BOOL ;	//S function 2 change
   S3Change : BOOL ;	//S function 3 change
   f60_3 : BOOL ;
   S1Quick : BOOL ;	//S function 1 quick
   S2Quick : BOOL ;	//S function 2 quick
   S3Quick : BOOL ;	//S function 3 quick
   f60_7 : BOOL ;
   T1Change : BOOL ;	//T function 1 change
   T2Change : BOOL ;	//T function 2 change
   T3Change : BOOL ;	//T function 3 change
   f61_3 : BOOL ;
   T1Quick : BOOL ;	//T function 1 quick
   T2Quick : BOOL ;	//T function 2 quick
   T3Quick : BOOL ;	//T function 3 quick
   f61_7 : BOOL ;
   D1Change : BOOL ;	//D function 1 change
   D2Change : BOOL ;	//D function 2 change
   D3Change : BOOL ;	//D function 3 change
   f62_3 : BOOL ;
   D1Quick : BOOL ;	//D function 1 quick
   D2Quick : BOOL ;	//D function 2 quick
   D3Quick : BOOL ;	//D function 3 quick
   f62_7 : BOOL ;
   EChange : BOOL ;	//E function change
   f63_1 : BOOL ;
   f63_2 : BOOL ;
   f63_3 : BOOL ;
   EQuick : BOOL ;	//E function quick
   f63_5 : BOOL ;
   f63_6 : BOOL ;
   f63_7 : BOOL ;
   H1Change : BOOL ;	//H function 1 change
   H2Change : BOOL ;	//H function 2 change
   H3Change : BOOL ;	//H function 3 change
   f64_3 : BOOL ;
   H1Quick : BOOL ;	//H function 1 quick
   H2Quick : BOOL ;	//H function 2 quick
   H3Quick : BOOL ;	//H function 3 quick
   f64_7 : BOOL ;
   F1Change : BOOL ;	//F function 1 change
   F2Change : BOOL ;	//F function 2 change
   F3Change : BOOL ;	//F function 3 change
   F4Change : BOOL ;	//F function 4 change
   F5Change : BOOL ;	//F function 5 change
   F6Change : BOOL ;	//F function 6 change
   f65_6 : BOOL ;
   f65_7 : BOOL ;
   M1Quick : BOOL ;	//M function 1 quick
   M2Quick : BOOL ;	//M function 2 quick
   M3Quick : BOOL ;	//M function 3 quick
   M4Quick : BOOL ;	//M function 4 quick
   M5Quick : BOOL ;	//M function 5 quick
   f66_5 : BOOL ;
   f66_6 : BOOL ;
   f66_7 : BOOL ;
   F1Quick : BOOL ;	//F function 1 quick
   F2Quick : BOOL ;	//F function 2 quick
   F3Quick : BOOL ;	//F function 3 quick
   F4Quick : BOOL ;	//F function 4 quick
   F5Quick : BOOL ;	//F function 5 quick
   F6Quick : BOOL ;	//F function 6 quick
   f67_6 : BOOL ;
   f67_7 : BOOL ;
   ExtM1 : INT ;	//Extended address M function 1 (16 bit INT)
   M1 : DINT ;	//M function 1 (DInt)
   ExtM2 : INT ;	//Extended address M function 1 (16 bit INT)
   M2 : DINT ;	//M function 2 (DInt)
   ExtM3 : INT ;	//Extended address M function 1 (16 bit INT)
   M3 : DINT ;	//M function 3 (DInt)
   ExtM4 : INT ;	//Extended address M function 1 (16 bit INT)
   M4 : DINT ;	//M function 4 (DInt)
   ExtM5 : INT ;	//Extended address M function 1 (16 bit INT)
   M5 : DINT ;	//M function 5 (DInt)
   ExtS1 : INT ;	//Extended address S function 1 (16 bit INT)
   S1 : REAL ;	//S function 1 (REAL)
   ExtS2 : INT ;	//Extended address S function 2 (16 bit INT)
   S2 : REAL ;	//S function 2 (REAL)
   ExtS3 : INT ;	//Extended address S function 3 (16 bit INT)
   S3 : REAL ;	//S function 3 (REAL)
   ExtT1 : INT ;	//Extended address T function 1 (16 bit INT)
//T : DINT; //T function (DInt)
//f122 :
   T1 : INT ;	//T function 1 (INT)
   ExtT2 : INT ;	//Extended address T function 2 (16 bit INT)
   T2 : INT ;	//T function 2 (INT)
   ExtT3 : INT ;	//Extended address T function 3 (16 bit INT)
   T3 : INT ;	//T function 3 (INT)
   ExtD1 : BYTE ;	//Extended address D function 1 (8 bit INT)
//D : INT;
//f132 : INT;   //Change in ca
   D1 : BYTE ;	//D function 1 (8 bit INT)
   ExtD2 : BYTE ;	//Extended address D function 2 (8 bit INT)
   D2 : BYTE ;	//D function 2 (8 bit INT)
   ExtD3 : BYTE ;	//Extended address D function 3 (8 bit INT)
   D3 : BYTE ;	//D function 3 (8 bit INT)
   ExtE : INT ;	//Extended address E function 3 (16 bit INT)
   E : REAL ;	//E function (REAL)
   ExtH1 : INT ;	//Extended address H function 1 (16 bit INT)
   H1 : REAL ;	//H function 1 (REAL)
   ExtH2 : INT ;	//Extended address H function 2 (16 bit INT)
   H2 : REAL ;	//H function 2 (REAL)
   ExtH3 : INT ;	//Extended address H function 3 (16 bit INT)
   H3 : REAL ;	//H function 3 (REAL)
   ExtF1 : INT ;	//Extended address F function 1 (16 bit INT)
   F1 : REAL ;	//F function 1 (REAL)
   ExtF2 : INT ;	//Extended address F function 2 (16 bit INT)
   F2 : REAL ;	//F function 2 (REAL)
   ExtF3 : INT ;	//Extended address F function 3 (16 bit INT)
   F3 : REAL ;	//F function 3 (REAL)
   ExtF4 : INT ;	//Extended address F function 4 (16 bit INT)
   F4 : REAL ;	//F function 4 (REAL)
   ExtF5 : INT ;	//Extended address F function 5 (16 bit INT)
   F5 : REAL ;	//F function 5 (REAL)
   ExtF6 : INT ;	//Extended address F function 6 (16 bit INT)
   F6 : REAL ;	//F function 6 (REAL)
   MDyn : ARRAY  [0 .. 99 ] OF BOOL ;	//Dynamic M functions [0..99]
   GAct : ARRAY  [1 .. 64 ] OF BYTE ;	//Active G function of group [1..64]
   E_MRPactivated : ARRAY  [1 .. 10 ] OF BOOL ;	//Machine-related protection area [1..10] preactivated
   E_CSPactivated : ARRAY  [1 .. 10 ] OF BOOL ;	//Channel-specific protection area [1..10] preactivated
   E_MRPViolated : ARRAY  [1 .. 10 ] OF BOOL ;	//Machine-related protection area [1..10] violated
   E_CSPViolated : ARRAY  [1 .. 10 ] OF BOOL ;	//Channel-specific protection area [1..10] violated
//from P4 on
   A_Str_DNo : BOOL ;	//Request of D number to NCK
   A_Str_Synon : BOOL ;	//Request of syn.action to NCK
   f_280_2 : BOOL ;
   f_280_3 : BOOL ;
   f_280_4 : BOOL ;
   f_280_5 : BOOL ;
   f_280_6 : BOOL ;
   f_280_7 : BOOL ;
   f_281_0 : BOOL ;
   A_Str_Synfrom : BOOL ;	//Request syn.action from NCK
   f_281_2 : BOOL ;
   f_281_3 : BOOL ;
   f_281_4 : BOOL ;
   f_281_5 : BOOL ;
   f_281_6 : BOOL ;
   f_281_7 : BOOL ;
   A_D1 : INT ;	//Assignment D1
   A_D2 : INT ;	//Assignment D2
   A_D3 : INT ;	//Assignment D3
   A_D4 : INT ;	//Assignment D4
   A_D5 : INT ;	//Assignment D5
   A_D6 : INT ;	//Assignment D6
   A_D7 : INT ;	//Assignment D7
   A_D8 : INT ;	//Assignment D8
   A_D9 : INT ;	//Assignment D9
   A_SynDisabl : ARRAY  [1 .. 64 ] OF BOOL ;	//Disable synchronous actions
   E_SynDisabled : ARRAY  [1 .. 64 ] OF BOOL ;	//Synchronous actions disabled
   E_G00 : BOOL ;	//Active G functions
   f316_1 : BOOL ;
   f316_2 : BOOL ;
   f316_3 : BOOL ;
   f316_4 : BOOL ;
   f316_5 : BOOL ;
   f316_6 : BOOL ;
   f316_7 : BOOL ;
   E_ExtLang : BOOL ;	// External language mode active
   E_WS_Setp : BOOL ;	// Workpiece setpoint reached
   f317_2 : BOOL ;
   f317_3 : BOOL ;
   f317_4 : BOOL ;
   E_DriveTest : BOOL ;	// Travel request drive test
   E_PTP_Travel : BOOL ;	//PTP travel active
   E_ToolMissing : BOOL ;	//Tool missing
   E_ASUP_Stop : BOOL ;	// ASUP stopped
   E_SearchAct : BOOL ;	// Search active
   E_TOFF : BOOL ;	// TOFF active
   E_TOFFmovem : BOOL ;	// TOFF movement active
   E_StopDelayed : BOOL ;	// Stop delayed
   E_AssM01 : BOOL ;	// Associated M01 active
   E_DRY : BOOL ;	// Dry-run feedrate active
   E_Overstore : BOOL ;	// Overstore active
   E_REPOS_EdgeAckn : BOOL ;	// REPOS MODE EDGE ACKN
   E_REPOS_PMode0 : BOOL ;	// Repos Path Mode Ackn 0
   E_REPOS_PMode1 : BOOL ;	// Repos Path Mode Ackn 0
   E_REPOS_PMode2 : BOOL ;	// Repos Path Mode Ackn 2
   E_DelayFTS : BOOL ;	// Delay FTS
   E_REPOS_DEFERRA : BOOL ;	// Repos DEFERRA L Chan
   E_Stop_NoDelayR : BOOL ;	// Stop-delayrange not activated
   E_NoToolChangeCmd : BOOL ;	// No tool change command active
   A_Ori : ARRAY  [1 .. 3 ] OF STRUCT 	//Control signals for orientation axes [1..3]
    HW_Bit0 : BOOL ;	//Activate handwheel Bit value coding
    HW_Bit1 : BOOL ;	//Activate handwheel Bit value coding
    HW_Bit2 : BOOL ;	//Activate handwheel Bit value coding
    FDStop : BOOL ;	//Feed stop
    Disabl : BOOL ;	//Traversing key disable
    RapidTrOR : BOOL ;	//Rapid traverse override
    Minus : BOOL ;	//Traversing key minus
    Plus : BOOL ;	//Traversing key plus
    INC1 : BOOL ;	//INC 1 active
    INC10 : BOOL ;	//INC 10 active
    INC100 : BOOL ;	//INC 100 active
    INC1000 : BOOL ;	//INC 1000 active
    INC10000 : BOOL ;	//INC 10000 active
    INCVar : BOOL ;	//INC variable active
    OEM : BYTE ;	//OEM signals
    InvHWDirOfRot : BOOL ;	// Inverting handwheel direction of rotation
    f3_1 : BOOL ;
    f3_2 : BOOL ;
    f3_3 : BOOL ;
    f3_4 : BOOL ;
    f3_5 : BOOL ;
    f3_6 : BOOL ;
    f3_7 : BOOL ;
   END_STRUCT ;
   E_Ori : ARRAY  [1 .. 3 ] OF STRUCT 	//Control signals for orientation axes [1..3]
    HW_Bit0 : BOOL ;	//Activate handwheel Bit value coding
    HW_Bit1 : BOOL ;	//Activate handwheel Bit value coding
    HW_Bit2 : BOOL ;	//Activate handwheel Bit value coding
    f0_3 : BOOL ;
    TReqMinus : BOOL ;	// Travel requests minus
    TReqPlus : BOOL ;	// Travel requests plus
    Minus : BOOL ;	//Traversing key minus
    Plus : BOOL ;	//Traversing key plus
    INC1 : BOOL ;	//INC 1 active
    INC10 : BOOL ;	//INC 10 active
    INC100 : BOOL ;	//INC 100 active
    INC1000 : BOOL ;	//INC 1000 active
    INC10000 : BOOL ;	//INC 10000 active
    INCVar : BOOL ;	//INC variable active
    OEM : BYTE ;	//OEM signals
    InvHWDirOfRot : BOOL ;	// Handwheel direction of rotation invert actively
    f3_1 : BOOL ;
    f3_2 : BOOL ;
    f3_3 : BOOL ;
    f3_4 : BOOL ;
    f3_5 : BOOL ;
    f3_6 : BOOL ;
    f3_7 : BOOL ;
   END_STRUCT ;
   E_T_PrewarnLimit : BOOL ;	//Tool prewarn limit reached
   E_T_Limit : BOOL ;	//Tool limit reached
   E_NewReplT : BOOL ;	//Transition to new replacement tool
   E_LastReplT : BOOL ;	//last replacement tool of the tool group
   f344_4 : BOOL ;
   f344_5 : BOOL ;
   f344_6 : BOOL ;
   f344_7 : BOOL ;
   f345 : BYTE ;
   f346 : BYTE ;
   f347 : BYTE ;
   E_T_NoPrewarnLimit : DINT ;	//T number for tool prewarn limit
   E_T_NoLimit : DINT ;	//T number for tool limit
   E_NewReplT_No : DINT ;	//T number of the new replacement tool
   E_LastReplT_No : DINT ;	//T number of the last replacement tool
   E_Cycle_Sig : ARRAY  [0 .. 15 ] OF BOOL ;	//Cycles Input Signals
   A_Cycle_Sig : ARRAY  [0 .. 15 ] OF BOOL ;	//Cycles Output Signals
   E_OEM_TechnoSig : ARRAY  [0 .. 31 ] OF BOOL ;	//OEM Techno Input Signals
   A_OEM_TechnoSig : ARRAY  [0 .. 31 ] OF BOOL ;	//OEM Techno Output Signals
   ProgEventDispl : BYTE ;	// ProgEventDisplay
   E_CollCheckStop : BOOL ;	// Stop of Collision Check
   E_StopCondition : BOOL ;	// Stop Condition
   f377_2 : BOOL ;
   f377_3 : BOOL ;
   E_JogRetract : BOOL ;	// JOG Retract active
   E_RetractData : BOOL ;	// Retract data available
   E_JOG_Circles : BOOL ;	// JOG in circles
   f377_7 : BOOL ;
   E_AnyAsup : BOOL ;	// AnyASUP activ
   E_SilentAsup : BOOL ;	// Silent ASUP activ
   f378_2 : BOOL ;
   f378_3 : BOOL ;
   f378_4 : BOOL ;
   f378_5 : BOOL ;
   f378_6 : BOOL ;
   f378_7 : BOOL ;
   f379 : BYTE ;
   f380 : ARRAY  [0 .. 31 ] OF BOOL ;	//Reserved
   A_ProgJump : BOOL ;	// control program jump
   f384_1 : BOOL ;
   f384_2 : BOOL ;
   f384_3 : BOOL ;
   f384_4 : BOOL ;
   f384_5 : BOOL ;
   f384_6 : BOOL ;
   f384_7 : BOOL ;
   f385 : BYTE ;
   f386 : WORD ;
   E_TransfoNo : BYTE ;	// active Transformation No.
   f389 : BYTE ;
   f390 : WORD ;
  END_STRUCT ;	
END_TYPE

